(* Logix 5000 project; controller CTRL_PLC_V30 vendor 1 type 14 code 212 rev 34.11; software revision 34.02 *)

TASK MainTask (continuous, watchdog 500 ms) : MainProgram, DataVersturen
TASK SafetyTask (periodic, rate 20 ms, priority 10, watchdog 20 ms, safety) : SafetyProgram

MODULES
   Local : vendor 1 type 14 code 212 (ICP 0, rev 34.11)
      PLC_ETH_CTRL : vendor 1 type 12 code 219 (Ethernet 192.168.1.120, ICP 2, rev 11.1)
      BUSPWR_CTRL : 2198-P208 (Ethernet 192.168.1.18, rev 14.1, A_MotionDiagnostics RPI 1 ms, B_MotionSync RPI 2 ms)
      DRIVER : vendor 1 type 45 code 12 (Ethernet 192.168.1.19, rev 9.3, C_Safety_Output RPI 20 ms, A_MotionDiagnostics RPI 1 ms, B_MotionSync RPI 2 ms, D_Safety_Input RPI 10 ms)
      RIO_CTRL : 1734-AENTR (Ethernet 192.168.1.113, rev 5.17, Output RPI 20 ms)
         Master_IOLINK : vendor 1 type 155 code 1 (PointIO 7, rev 2.1, StandardDataDriven RPI 20 ms)   // 4 channel master IO-link
         INP1_CTRL : 1734-IB4 (PointIO 3, rev 3.1)
         INP2_CTRL : 1734-IB4 (PointIO 4, rev 3.1)
         OUTP2_CTRL : vendor 1 type 7 code 231 (PointIO 6, rev 3.1)
         OUTP1_CTRL : vendor 1 type 7 code 231 (PointIO 5, rev 3.1)
         Safety_OUT : vendor 1 type 35 code 16 (PointIO 2, rev 2.1, Output RPI 20 ms, Input RPI 10 ms)
         Safety_IN : vendor 1 type 35 code 15 (PointIO 1, rev 2.1, Output RPI 20 ms, Input RPI 10 ms)
      @fcc730f7@:Partner : vendor 1 type 14 code 171 (ICP 1, rev 34.11)
END_MODULES

TYPE UDT_COMM_CTRL_TO_SPLC :
STRUCT
   CONTROLLER_STATUS : CONNECTION_STATUS;
   AUX_MCHS_WATCHDOG_CC_BT : BOOL;
   CMD_CCMN_SCLW_RAD_RELEASE_BRAKE : BOOL;
   CMD_CCMN_SWRW_RAD_RELEASE_BRAKE : BOOL;
   CMD_TEST_ABSR_MODULE : BOOL;
   CMD_TEST_ACSR_MODULE : BOOL;
   CMD_TEST_CHAF_MODULE : BOOL;
   CMD_TEST_MODULAR : BOOL;
   CMD_TEST_RBOT_MODULE : BOOL;
   CMD_TEST_RSSR_MODULE : BOOL;
   CMD_TEST_SARB_MODULE : BOOL;
   CMD_TEST_SWSR_MODULE : BOOL;
   CMD_TEST_TBM_MODULE : BOOL;
   QSP_BTDS_XBTDS_DISABLE_LIMITS : BOOL;
   QSP_CCMB_LASERLIGHT_ON : BOOL;
   QSP_CCMF_LASERLIGHT_ON : BOOL;
   QSP_GTCV_ACKNOWLEDGE_MUTE_SCREEN : BOOL;
   QSP_GTRU_TRAV_TO_PICKUP : BOOL;
   QSP_GTRU_TRAV_TO_RELEASE : BOOL;
   QSP_XBDSL_FEEDBACK_FAULT_BRAKE : BOOL;
   QSP_XBDSR_FEEDBACK_FAULT_BRAKE : BOOL;
   QSP_XBTDS_FEEDBACK_FAULT_BRAKE : BOOL;
   QSP_XCCDS_FEEDBACK_FAULT_BRAKE : BOOL;
   QSP_XPBST_FEEDBACK_FAULT_BRAKE : BOOL;
   ZZZ_CC_TO_BT_BOOL_1 : BOOL;
   ZZZ_CC_TO_BT_BOOL_2 : BOOL;
   ZZZ_CC_TO_BT_BOOL_3 : BOOL;
   ZZZ_CC_TO_BT_BOOL_4 : BOOL;
   ZZZ_CC_TO_BT_BOOL_5 : BOOL;
   ZZZ_CC_TO_BT_BOOL_6 : BOOL;
   ZZZ_CC_TO_BT_BOOL_7 : BOOL;
   ZZZ_CC_TO_BT_BOOL_8 : BOOL;
   ZZZ_CC_TO_BT_BOOL_9 : BOOL;
   ZZZ_CC_TO_BT_REAL_1 : REAL;
   ZZZ_CC_TO_BT_REAL_2 : REAL;
   ZZZ_CC_TO_BT_REAL_3 : REAL;
   ZZZ_CC_TO_BT_REAL_4 : REAL;
   ZZZ_CC_TO_BT_REAL_5 : REAL;
END_STRUCT
END_TYPE

TYPE UDT_COMM_SPLC_TO_CTRL :
STRUCT
   CONTROLLER_STATUS : CONNECTION_STATUS;
   AUX_MCHS_WATCHDOG_BT_CC : BOOL;
   CMD_SPLC_IFS_CCAM_STEP_TBM : BOOL;
   FATAL_FAULTS_HWDI : DINT;
   FATAL_FAULTS_HWDI_SIO : DINT;
   FATAL_FAULTS_MCHG : DINT;
   FATAL_FAULTS_MCHS : DINT;
   FATAL_FAULTS_SPLC_ABSR : DINT;
   FATAL_FAULTS_SPLC_ACSR : DINT;
   FATAL_FAULTS_SPLC_BDST : DINT;
   FATAL_FAULTS_SPLC_RSSR : DINT;
   FATAL_FAULTS_SPLC_SARB : DINT;
   FATAL_FAULTS_SPLC_SCCV : DINT;
   FATAL_FAULTS_SPLC_SWSR : DINT;
   FATAL_FAULTS_SPLC_TBM : DINT;
   FCO_HWDI_SYSTEMS_OK_SPLC : BOOL;
   ICF_SPLC_BEAM22_PRESENT : BOOL;
   ICF_SPLC_ROBOT_PREPARED : BOOL;
   ICR_BTDS_NOT_AT_LEFT_POS_LIMIT : BOOL;
   ICR_BTDS_NOT_AT_RIGHT_NEG_LIMIT : BOOL;
   ICR_BTMO_MOTORS_OFF_FEEDBACK : BOOL;
   ICR_CCDS_NOT_AT_LEFT_NEG_LIMIT : BOOL;
   ICR_CCDS_NOT_AT_RIGHT_POS_LIMIT : BOOL;
   IFS_BSMN_1BL2_REWIND_MATERIAL : BOOL;
   IFS_BSMN_1BLO_REWIND_MATERIAL : BOOL;
   IFS_BSMN_2BL2_REWIND_MATERIAL : BOOL;
   IFS_BSMN_2BLO_REWIND_MATERIAL : BOOL;
   IFS_BTAM_STEP : BOOL;
   IFS_CCAM_STEP : BOOL;
   IFS_CSMN_1PLO_REWIND_MATERIAL : BOOL;
   IFS_CSMN_2PLO_REWIND_MATERIAL : BOOL;
   IFS_CSMN_3PLO_REWIND_MATERIAL : BOOL;
   IFS_CSMN_INLO_REWIND_MATERIAL : BOOL;
   IKS_MCHG_CONTROLS_ON : BOOL;
   IPB_BSMN_1BL2_CNV_FEED2 : BOOL;
   IPB_BSMN_2BL2_CNV_FEED : BOOL;
   IPB_CSMN_INCV_FEED_INSIDE : BOOL;
   IPB_CSMN_SWLO_LFT_CNV_FEED2 : BOOL;
   ISP_1BAR_CONNECT_MOTORS : BOOL;
   ISP_1BAR_DRIVE_ENABLE : BOOL;
   ISP_1BCU_SAFETY_DOORS_CLOSED : BOOL;
   ISP_1BCV_CONNECT_MOTORS : BOOL;
   ISP_1BCV_DRIVE_ENABLE : BOOL;
   ISP_1BL2_SAFETY_NOT_ACTIVATED : BOOL;
   ISP_1BLO_SAFETY_NOT_ACTIVATED : BOOL;
   ISP_1PCV_CONNECT_MOTORS : BOOL;
   ISP_1PCV_DRIVE_ENABLE : BOOL;
   ISP_1PLO_SAFETY_NOT_ACTIVATED : BOOL;
   ISP_2BAR_CONNECT_MOTORS : BOOL;
   ISP_2BAR_DRIVE_ENABLE : BOOL;
   ISP_2BCU_SAFETY_DOORS_CLOSED : BOOL;
   ISP_2BCV_CONNECT_MOTORS : BOOL;
   ISP_2BCV_DRIVE_ENABLE : BOOL;
   ISP_2BL2_SAFETY_NOT_ACTIVATED : BOOL;
   ISP_2BLO_SAFETY_NOT_ACTIVATED : BOOL;
   ISP_2PCV_CONNECT_MOTORS : BOOL;
   ISP_2PCV_DRIVE_ENABLE : BOOL;
   ISP_3PCV_CONNECT_MOTORS : BOOL;
   ISP_3PCV_DRIVE_ENABLE : BOOL;
   ISP_2PLO_SAFETY_NOT_ACTIVATED : BOOL;
   ISP_3PLO_SAFETY_NOT_ACTIVATED : BOOL;
   ISP_BDLD_CONNECT_MOTORS : BOOL;
   ISP_BDLD_DRIVE_ENABLE : BOOL;
   ISP_BDLD_LIGHT_CURTAIN_BLOCKED : BOOL;
   ISP_BDLD_RAD_AT_FRONT : BOOL;
   ISP_BDLD_RAD_AT_FRONT_SAFE_AREA : BOOL;
   ISP_BDLD_RAD_AT_MIDDLE : BOOL;
   ISP_BDLD_SAFETY_NOT_ACTIVATED : BOOL;
   ISP_BDSE_INITIALIZE_ARMS : BOOL;
   ISP_BDSE_LFT_CONNECT_MOTORS : BOOL;
   ISP_BDSE_LFT_DRIVE_ENABLE : BOOL;
   ISP_BDSE_RHT_AT_LOAD_AREA : BOOL;
   ISP_BDSE_RHT_CONNECT_MOTORS : BOOL;
   ISP_BDSE_RHT_DRIVE_ENABLE : BOOL;
   ISP_BDST_LOAD_SAFETY_SCR_NOT_TRIPPED : BOOL;
   ISP_BDST_MID_SAFETY_SCR_NOT_TRIPPED : BOOL;
   ISP_BDST_REAR_SAFETY_SCR_NOT_TRIPPED : BOOL;
   ISP_BDST_REAR_SAFETY_SCR_OK : BOOL;
   ISP_BPCA_CONNECT_MOTORS : BOOL;
   ISP_BPCA_DRIVE_ENABLE : BOOL;
   ISP_BPCU_SAFETY_DOOR_CLOSED : BOOL;
   ISP_BPCU_SAFETY_FENCES_CLOSED : BOOL;
   ISP_BPCV_CONNECT_MOTORS : BOOL;
   ISP_BPCV_DRIVE_ENABLE : BOOL;
   ISP_BPSO_CONNECT_MOTORS : BOOL;
   ISP_BPSO_DRIVE_ENABLE : BOOL;
   ISP_BSCV_CONNECT_MOTORS : BOOL;
   ISP_BSCV_DRIVE_ENABLE : BOOL;
   ISP_BTDD_CONNECT_MOTORS : BOOL;
   ISP_BTDD_DRIVE_ENABLE : BOOL;
   ISP_BTDD_RELEASE_BRAKE : BOOL;
   ISP_BTDH_CONNECT_MOTORS : BOOL;
   ISP_BTDH_DRIVE_ENABLE : BOOL;
   ISP_BTDH_RELEASE_BRAKE : BOOL;
   ISP_BTDR_CONNECT_MOTORS : BOOL;
   ISP_BTDR_DRIVE_ENABLE : BOOL;
   ISP_BTDR_RELEASE_BRAKE : BOOL;
   ISP_BTDS_AT_BTTR_AREA : BOOL;
   ISP_BTDS_CONNECT_MOTORS : BOOL;
   ISP_BTDS_DRIVE_ENABLE : BOOL;
   ISP_BTDS_LEFT_LIMIT_OK : BOOL;
   ISP_BTDS_RIGHT_LIMIT_OK : BOOL;
   ISP_BTMN_AREA_ENTRY_NOT_ACTIVE : BOOL;
   ISP_BTMN_BT_DRUM_REL_BRAKE_MODE_ACTIVE : BOOL;
   ISP_BTMN_DOOR_TBM_BR1_SAFETY_NOT_TRIPPED : BOOL;
   ISP_BTMN_DOOR_TBM_BR2_SAFETY_NOT_TRIPPED : BOOL;
   ISP_BTMN_LFT_TRACK_FIRST_RESET_DONE : BOOL;
   ISP_BTMN_LFT_TRACK_SAFETY_NOT_ACTIVATED : BOOL;
   ISP_BTMN_REAR_TRACK_FIRST_RESET_DONE : BOOL;
   ISP_BTMN_REAR_TRACK_SAF_NOT_ACTIVATED : BOOL;
   ISP_BTMN_RHT_TRACK_SAFETY_NOT_ACTIVATED : BOOL;
   ISP_BTMN_TBM_AREA_NOT_ACTIVATED : BOOL;
   ISP_BTMN_TBM_BT_JOG_MODE : BOOL;
   ISP_BTMN_TBM_BT_SHUTTLE_REL_BRAKE_MODE : BOOL;
   ISP_BTMO_RAD_DRIVE_ENABLE : BOOL;
   ISP_BTMO_SAFETY_OVERRULED : BOOL;
   ISP_CCDR_CDAR_CONNECT_MOTORS : BOOL;
   ISP_CCDR_CDRO_CONNECT_MOTORS : BOOL;
   ISP_CCDR_CDTR_CONNECT_MOTORS : BOOL;
   ISP_CCDS_AT_ACSR_POSITION : BOOL;
   ISP_CCDS_CONNECT_MOTORS : BOOL;
   ISP_CCDS_DRIVE_ENABLE : BOOL;
   ISP_CCDS_LEFT_LIMIT_OK : BOOL;
   ISP_CCDS_RIGHT_LIMIT_OK : BOOL;
   ISP_CCMB_SAFETY_OVERRULED : BOOL;
   ISP_CCMC_DRIVE_ENABLE : BOOL;
   ISP_CCMF_CONNECT_MOTORS : BOOL;
   ISP_CCMF_SAFETY_OVERRULED : BOOL;
   ISP_CCMN_BDLD_AREA_NOT_ACTIVATED : BOOL;
   ISP_CCMN_DOOR_TBM_REAR_SAF_NOT_TRIPPED : BOOL;
   ISP_CCMN_FRNT_TRACK_SAFETY_NOT_ACTIVATED : BOOL;
   ISP_CCMN_OPERATOR_AREA_ENTRY_NOT_ACTIVE : BOOL;
   ISP_CCMN_OPERATOR_AREA_NOT_ACTIVATED : BOOL;
   ISP_CCMN_REAR_TRACK_FIRST_RESET_DONE : BOOL;
   ISP_CCMN_REAR_TRACK_SAF_NOT_ACTIVATED : BOOL;
   ISP_CCMN_TBM_AREA_ENTRY_NOT_ACTIVE : BOOL;
   ISP_CCMN_TBM_AREA_NOT_ACTIVATED : BOOL;
   ISP_CCMN_TBM_CC_JOG_MODE : BOOL;
   ISP_CCMN_TBM_CC_SHUTTLE_REL_BRAKE_MODE : BOOL;
   ISP_CCMR_DRIVE_ENABLE : BOOL;
   ISP_CCMT_DRIVE_ENABLE : BOOL;
   ISP_CDAR_DRIVE_ENABLE : BOOL;
   ISP_CDRO_DRIVE_ENABLE : BOOL;
   ISP_CDTR_DRIVE_ENABLE : BOOL;
   ISP_CENT_BT_SAFETY_OK : BOOL;
   ISP_CENT_CC_SAFETY_OK : BOOL;
   ISP_CWLO_FEST_SAFETY_DOOR_CLOSED : BOOL;
   ISP_CWLO_LFT_STRIP_NOT_SELECTED : BOOL;
   ISP_CWLO_RHT_STRIP_NOT_SELECTED : BOOL;
   ISP_CWLO_SAFETY_DOOR_CLOSED : BOOL;
   ISP_CWTC_CONNECT_MOTORS : BOOL;
   S_ISP_CWTC_DRIVE_ENABLE : BOOL;
   ISP_E_STOP_ACTIVATED : BOOL;
   ISP_GTCV_EJECTION_TABLE_UP : BOOL;
   ISP_GTRU_CONNECT_MOTORS : BOOL;
   ISP_GTRU_DRIVE_ENABLE : BOOL;
   ISP_GTRU_GRIPPER_OPEN : BOOL;
   ISP_GTRU_LIGHT_CURTAIN_BLOCKED : BOOL;
   ISP_GTRU_RAD_AT_FRONT : BOOL;
   ISP_GTRU_SAFETY_MUTE_ACTIVE : BOOL;
   ISP_GTRU_SAFETY_NOT_ACTIVATED : BOOL;
   ISP_GTRU_TIRE_DETECTED : BOOL;
   ISP_GTRU_TRAV_AT_PICKUP : BOOL;
   ISP_GTRU_TRAV_AT_RELEASE : BOOL;
   ISP_INCV_CONNECT_MOTORS : BOOL;
   ISP_INCV_DRIVE_ENABLE : BOOL;
   ISP_INLO_SAFETY_NOT_ACTIVATED : BOOL;
   ISP_MAIN_PRESSURE_PRESENT : BOOL;
   ISP_PACU_SAFETY_DOOR_CLOSED : BOOL;
   ISP_PACU_SAFETY_FENCES_CLOSED : BOOL;
   ISP_PACV_CONNECT_MOTORS : BOOL;
   ISP_PACV_DRIVE_ENABLE : BOOL;
   ISP_PBCV_CONNECT_MOTORS : BOOL;
   ISP_PBCV_DRIVE_ENABLE : BOOL;
   ISP_PBCV_SAFETY_DOORS_CLOSED : BOOL;
   ISP_PBST_CONNECT_MOTORS : BOOL;
   ISP_PBST_DRIVE_ENABLE : BOOL;
   ISP_PBUD_CONNECT_MOTORS : BOOL;
   ISP_PBUD_DRIVE_ENABLE : BOOL;
   ISP_PBUD_SAFE_SPD_TRIPPED : BOOL;
   ISP_RBCL_CONNECT_MOTORS : BOOL;
   ISP_RBCL_DRIVE_ENABLE : BOOL;
   ISP_RBOT_ENABLE : BOOL;
   ISP_RSLC_CONNECT_MOTORS : BOOL;
   ISP_RSLC_DRIVE_ENABLE : BOOL;
   ISP_RSLO_REAR_SAFETY_NOT_ACTIVATED : BOOL;
   ISP_RSLO_SIDE_SAFETY_NOT_ACTIVATED : BOOL;
   ISP_RSLW_AT_LETOFF_AREA : BOOL;
   ISP_RSLW_CONNECT_MOTORS : BOOL;
   ISP_RSLW_DRIVE_ENABLE : BOOL;
   ISP_RSLW_RAD_CONNECT_MOTORS : BOOL;
   ISP_RSLW_RAD_DRIVE_ENABLE : BOOL;
   ISP_RSLW_TRAV_CONNECT_MOTORS : BOOL;
   ISP_RSLW_TRAV_DRIVE_ENABLE : BOOL;
   ISP_RSMN_JOG_MODE : BOOL;
   ISP_RSMN_RS_INSIDE_FIRST_RESET_DONE : BOOL;
   ISP_RSMN_RSLO_JOG_MODE : BOOL;
   ISP_RSMN_RSLO_LFT_JOG_MODE : BOOL;
   ISP_RSMN_RSLO_RHT_JOG_MODE : BOOL;
   ISP_RSMN_RSXR_REL_BRAKE_MODE : BOOL;
   ISP_RSMN_TBM_AREA_SAFETY_NOT_ACTIVE : BOOL;
   ISP_RSRC_CONNECT_MOTORS : BOOL;
   ISP_RSRC_DRIVE_ENABLE : BOOL;
   ISP_RSRW_CONNECT_MOTORS : BOOL;
   ISP_RSRW_DRIVE_ENABLE : BOOL;
   ISP_RSRW_RAD_CONNECT_MOTORS : BOOL;
   ISP_RSRW_RAD_DRIVE_ENABLE : BOOL;
   ISP_RSRW_TRAV_CONNECT_MOTORS : BOOL;
   ISP_RSRW_TRAV_DRIVE_ENABLE : BOOL;
   ISP_SARB_ENABLE : BOOL;
   ISP_SCLW_AT_LETOFF_AREA : BOOL;
   ISP_SCLW_CONNECT_MOTORS : BOOL;
   ISP_SCLW_DRIVE_ENABLE : BOOL;
   ISP_SCLW_RAD_CONNECT_MOTORS : BOOL;
   ISP_SCLW_RAD_DRIVE_ENABLE : BOOL;
   ISP_SCLW_TRAV_CONNECT_MOTORS : BOOL;
   ISP_SCLW_TRAV_DRIVE_ENABLE : BOOL;
   ISP_SCMN_JOG_MODE : BOOL;
   ISP_SCMN_RELEASE_SCXR_BRAKE : BOOL;
   ISP_SCMN_SC_INSIDE_FIRST_RESET_DONE : BOOL;
   ISP_SCMN_TBM_AREA_SAFETY_NOT_ACTIVE : BOOL;
   ISP_SCRW_CONNECT_MOTORS : BOOL;
   ISP_SCRW_DRIVE_ENABLE : BOOL;
   ISP_SCRW_RAD_CONNECT_MOTORS : BOOL;
   ISP_SCRW_RAD_DRIVE_ENABLE : BOOL;
   ISP_SCRW_TRAV_CONNECT_MOTORS : BOOL;
   ISP_SCRW_TRAV_DRIVE_ENABLE : BOOL;
   ISP_SLOW_START_PRESSURE_NOT_OK : BOOL;
   ISP_SPLC_FAULT_EXISTS : BOOL;
   ISP_SPLC_REAR_TRACK_SAFETY_RST_INITIATED : BOOL;
   ISP_SPLC_SAFETY_SIGNATURE_EXISTS : BOOL;
   ISP_SPLC_TBM_BT_AREA_ENTRY_OK_DELAY : BOOL;
   ISP_SPLC_TBM_BT_LC_OK_DELAY : BOOL;
   ISP_SPLC_TBM_CC_AREA_ENTRY_OPER_OK_DELAY : BOOL;
   ISP_SPLC_TBM_CC_AREA_ENTRY_TBM_OK_DELAY : BOOL;
   ISP_SPLC_TBM_CC_LC_OPER_OK_DELAY : BOOL;
   ISP_SPLC_TBM_CC_LC_TBM_OK_DELAY : BOOL;
   ISP_SWL2_SAFETY_NOT_ACTIVATED : BOOL;
   ISP_SWL3_REAR_SAFETY_NOT_ACTIVATED : BOOL;
   ISP_SWL3_SIDE_SAFETY_NOT_ACTIVATED : BOOL;
   ISP_SWLC_CONNECT_MOTORS : BOOL;
   ISP_SWLC_DRIVE_ENABLE : BOOL;
   ISP_SWLO_INSIDE_SAFETY_NOT_ACTIVE : BOOL;
   ISP_SWLO_SAFETY_NOT_ACTIVATED : BOOL;
   ISP_SWLW_AT_LETOFF_AREA : BOOL;
   ISP_SWLW_CONNECT_MOTORS : BOOL;
   ISP_SWLW_DRIVE_ENABLE : BOOL;
   ISP_SWLW_RAD_CONNECT_MOTORS : BOOL;
   ISP_SWLW_RAD_DRIVE_ENABLE : BOOL;
   ISP_SWLW_TRAV_CONNECT_MOTORS : BOOL;
   ISP_SWLW_TRAV_DRIVE_ENABLE : BOOL;
   ISP_SWMN_JOG_MODE : BOOL;
   ISP_SWMN_SW_INSIDE_FIRST_RESET_DONE : BOOL;
   ISP_SWMN_SWL3_JOG_MODE : BOOL;
   ISP_SWMN_SWL3_LFT_JOG_MODE : BOOL;
   ISP_SWMN_SWL3_RHT_JOG_MODE : BOOL;
   ISP_SWMN_SWLC_DOOR_CLOSED : BOOL;
   ISP_SWMN_RELEASE_SWXR_BRAKE : BOOL;
   ISP_SWMN_TBM_AREA_SAFETY_NOT_ACTIVE : BOOL;
   ISP_SWRC_CONNECT_MOTORS : BOOL;
   ISP_SWRC_DRIVE_ENABLE : BOOL;
   ISP_SWRW_CONNECT_MOTORS : BOOL;
   ISP_SWRW_DRIVE_ENABLE : BOOL;
   ISP_SWRW_RAD_CONNECT_MOTORS : BOOL;
   ISP_SWRW_RAD_DRIVE_ENABLE : BOOL;
   ISP_SWRW_TRAV_CONNECT_MOTORS : BOOL;
   ISP_SWRW_TRAV_DRIVE_ENABLE : BOOL;
   ISP_TDAR_CONNECT_MOTORS : BOOL;
   ISP_TDAR_DRIVE_ENABLE : BOOL;
   ISP_TDCU_SAFETY_COVER_CLOSED : BOOL;
   ISP_TDCV_CONNECT_MOTORS : BOOL;
   ISP_TDCV_DRIVE_ENABLE : BOOL;
   ISP_TDLO_LFT_SAFETY_NOT_ACTIVATED : BOOL;
   ISP_TDLO_RHT_SAFETY_NOT_ACTIVATED : BOOL;
   ISP_TDLO_SAFETY_NOT_ACTIVATED : BOOL;
   ISP_TEST_MODE_SELECTED : BOOL;
   ISP_TPGU_SAFETY_OVERRULED : BOOL;
   ISS_BSMN_1BL2_WINDOFF : BOOL;
   ISS_BSMN_1BL2_WINDUP : BOOL;
   ISS_BSMN_1BLO_WINDOFF : BOOL;
   ISS_BSMN_1BLO_WINDUP : BOOL;
   ISS_BSMN_2BL2_WINDOFF : BOOL;
   ISS_BSMN_2BL2_WINDUP : BOOL;
   ISS_BSMN_2BLO_WINDOFF : BOOL;
   ISS_BSMN_2BLO_WINDUP : BOOL;
   ISS_CSMN_1PLO_WINDOFF : BOOL;
   ISS_CSMN_1PLO_WINDUP : BOOL;
   ISS_CSMN_2PLO_WINDOFF : BOOL;
   ISS_CSMN_2PLO_WINDUP : BOOL;
   ISS_CSMN_3PLO_WINDOFF : BOOL;
   ISS_CSMN_3PLO_WINDUP : BOOL;
   ISS_CSMN_INLO_WINDOFF : BOOL;
   ISS_CSMN_INLO_WINDUP : BOOL;
   ISS_CSMN_SWL2_LFT_WINDOFF : BOOL;
   ISS_CSMN_SWL2_LFT_WINDUP : BOOL;
   ISS_CSMN_SWL2_RHT_WINDOFF : BOOL;
   ISS_CSMN_SWL2_RHT_WINDUP : BOOL;
   ISS_CSMN_SWL2_WINDOFF : BOOL;
   ISS_CSMN_SWL2_WINDUP : BOOL;
   ISS_CSMN_SWLO_LFT_WINDOFF : BOOL;
   ISS_CSMN_SWLO_LFT_WINDUP : BOOL;
   ISS_CSMN_SWLO_RHT_WINDOFF : BOOL;
   ISS_CSMN_SWLO_RHT_WINDUP : BOOL;
   ISS_CSMN_SWLO_WINDOFF : BOOL;
   ISS_CSMN_SWLO_WINDUP : BOOL;
   ISS_RSMN_RSLW_JOG_FWD : BOOL;
   ISS_RSMN_RSLW_JOG_REV : BOOL;
   ISS_RSMN_RSRW_JOG_FWD : BOOL;
   ISS_RSMN_RSRW_JOG_REV : BOOL;
   ISS_SCMN_SCLW_JOG_FWD : BOOL;
   ISS_SCMN_SCLW_JOG_REV : BOOL;
   ISS_SCMN_SCRW_JOG_FWD : BOOL;
   ISS_SCMN_SCRW_JOG_REV : BOOL;
   ISS_SWMN_SWLW_JOG_FWD : BOOL;
   ISS_SWMN_SWLW_JOG_REV : BOOL;
   ISS_SWMN_SWRW_JOG_FWD : BOOL;
   ISS_SWMN_SWRW_JOG_REV : BOOL;
   ISS_TDMN_TDLO_LFT_WINDOFF : BOOL;
   ISS_TDMN_TDLO_LFT_WINDUP : BOOL;
   ISS_TDMN_TDLO_RHT_WINDOFF : BOOL;
   ISS_TDMN_TDLO_RHT_WINDUP : BOOL;
   ISS_TDMN_TDLO_WINDOFF : BOOL;
   ISS_TDMN_TDLO_WINDUP : BOOL;
   ISP_XXMN_DOOR_ACSR_XX_CLOSED : BOOL;
   ISP_XXMN_DOOR_SC_XX_CLOSED : BOOL;
   ISP_XXMN_DOOR_XX_TBM_CLOSED : BOOL;
   ISP_XXMN_INSIDE_SAFETY_BTTR_RESET_REQ : BOOL;
   ZZZ_BT_TO_CC_BOOL_1 : BOOL;
   ZZZ_BT_TO_CC_BOOL_2 : BOOL;
   ZZZ_BT_TO_CC_BOOL_3 : BOOL;
   ZZZ_BT_TO_CC_BOOL_4 : BOOL;
   ZZZ_BT_TO_CC_BOOL_5 : BOOL;
   ZZZ_BT_TO_CC_BOOL_6 : BOOL;
   ZZZ_BT_TO_CC_BOOL_7 : BOOL;
   ZZZ_BT_TO_CC_BOOL_8 : BOOL;
   ZZZ_BT_TO_CC_BOOL_9 : BOOL;
   ZZZ_BT_TO_CC_REAL_1 : REAL;
   ZZZ_BT_TO_CC_REAL_2 : REAL;
   ZZZ_BT_TO_CC_REAL_3 : REAL;
   ZZZ_BT_TO_CC_REAL_4 : REAL;
   ZZZ_BT_TO_CC_REAL_5 : REAL;
   ISS_BSMN_1BLO_DRIVE_ROLLS_TO_REST : BOOL;
   ISS_BSMN_1BLO_DRIVE_ROLLS_ENGAGE : BOOL;
   ISP_1BLO_TWO_HAND_OVERRIDE : BOOL;
   ISS_BSMN_1BLO_CART_LOCK : BOOL;
   ISS_BSMN_1BLO_CART_UNLOCK : BOOL;
   ISS_BSMN_2BLO_DRIVE_ROLLS_TO_REST : BOOL;
   ISS_BSMN_2BLO_DRIVE_ROLLS_ENGAGE : BOOL;
   ISP_2BLO_TWO_HAND_OVERRIDE : BOOL;
   ISS_BSMN_2BLO_CART_LOCK : BOOL;
   ISS_BSMN_2BLO_CART_UNLOCK : BOOL;
   ISS_TDMN_TDLO_DRIVE_ROLLS_ENGAGE : BOOL;
   ISS_TDMN_TDLO_DRIVE_ROLLS_TO_REST : BOOL;
   ISP_TDLO_TWO_HAND_OVERRIDE : BOOL;
   ISS_TDMN_TDLO_CART_LOCK : BOOL;
   ISS_TDMN_TDLO_CART_UNLOCK : BOOL;
   ISS_SWLO_RHT_DRIVE_ROLLS_REST : BOOL;
   ISS_SWLO_RHT_DRIVE_ROLLS_ENGAGE : BOOL;
   ISS_CSMN_SWLO_RHT_CART_LOCK : BOOL;
   ISS_CSMN_SWLO_RHT_CART_UNLOCK : BOOL;
   ISP_SWLO_RHT_TWO_HAND_OVERRIDE : BOOL;
   ISS_SWLO_LFT_DRIVE_ROLLS_REST : BOOL;
   ISS_SWLO_LFT_DRIVE_ROLLS_ENGAGE : BOOL;
   ISS_CSMN_SWLO_LFT_CART_LOCK : BOOL;
   ISS_CSMN_SWLO_LFT_CART_UNLOCK : BOOL;
   ISP_SWLO_LFT_TWO_HAND_OVERRIDE : BOOL;
END_STRUCT
END_TYPE

VAR_GLOBAL   (* controller tags *)
   Aantal_RondjesT1 : DINT := 40;
   Aantal_RondjesT2 : DINT;
   As_Test1_CTRL : AXIS_CIP_DRIVE;
   As_Test2_CTRL : AXIS_CIP_DRIVE;
   AsTest1Accel : REAL := 1000000.0;
   AsTest1Snelheid : REAL := 3500.0;
   AsTest1StartPos : REAL;
   AsTest1StopPos : REAL := 9500.0;
   AsTest2Accel : REAL;
   AsTest2Snelheid : REAL;
   AsTest2StartPos : REAL;
   AsTest2StopPos : REAL;
   BOOL : BOOL;
   Control_Volt_Van_SAF : BOOL;
   Drive1 : MOTION_GROUP;
   Drive_SAFE_OFF1 : ALIAS FOR DRIVER:SO.SafeTorqueOff1;
   Drive_SAFE_OFF2 : ALIAS FOR DRIVER:SO.SafeTorqueOff2;
   ERROR : BOOL;
   ERROR_1 : BOOL := 1;
   ERROR_2 : BOOL := 1;
   ESTP_ACTIVATED : BOOL;
   HomeT1 : ALIAS FOR IOP_HMI_BT[0].2;
   HomeT2 : ALIAS FOR IOP_HMI_BT[1].2;
   ILB_RESET_SAFETY1 : BOOL := 1;
   ILG_CTRL_VOLT1 : BOOL;
   IO_CTRL_TO_SPLC : UDT_COMM_CTRL_TO_SPLC := (CONTROLLER_STATUS.RunMode := 1); {produced}
   IO_SPLC_TO_CTRL : UDT_COMM_SPLC_TO_CTRL;
   IOP_HMI_BT : DINT[2];
   IOP_HMI_REAL : REAL[20] := ([0] := 3500.0, [1] := 1000000.0, [3] := 9500.0, [4] := 40.0);
   MDA_DATACHOICE : INT := 2;
   MDB_DATACHOICE : INT := 2;
   Motionback : MOTION_INSTRUCTION;
   Motionback2 : MOTION_INSTRUCTION;
   Motioncontrol13 : MOTION_INSTRUCTION := (FLAGS := -1845493760, EN := 1, ER := 1, ERR := 13, EXERR := 6);
   Motioncontrol14 : MOTION_INSTRUCTION := (FLAGS := -1845493760, EN := 1, ER := 1, ERR := 13, EXERR := 6);
   Motioncontrol20 : MOTION_INSTRUCTION;
   Motioncontrol21 : MOTION_INSTRUCTION := (FLAGS := -1476395008, EN := 1, DN := 1, PC := 1, STATE := 17);
   Motioncontrol26 : MOTION_INSTRUCTION := (FLAGS := -1442840576, EN := 1, DN := 1, PC := 1, STATE := 17); {access None}
   Motioncontrol27 : MOTION_INSTRUCTION := (FLAGS := -1442840576, EN := 1, DN := 1, PC := 1, STATE := 17);
   Motioncontrol3 : MOTION_INSTRUCTION := (FLAGS := -1442840576, EN := 1, DN := 1, PC := 1);
   Motioncontrol30 : MOTION_INSTRUCTION := (FLAGS := 33554432);
   Motioncontrol31 : MOTION_INSTRUCTION;
   Motioncontrol4 : MOTION_INSTRUCTION := (FLAGS := -1442840576, EN := 1, DN := 1, PC := 1);
   Motionctrl1 : MOTION_INSTRUCTION := (FLAGS := -1577058304, EN := 1, DN := 1, STATE := 1);
   Motionctrl2 : MOTION_INSTRUCTION := (FLAGS := -1577058304, EN := 1, DN := 1, STATE := 1);
   Motionstart1 : MOTION_INSTRUCTION := (FLAGS := -1845493760, EN := 1, ER := 1, ERR := 20);
   Motionstartl2 : MOTION_INSTRUCTION := (FLAGS := -1845493760, EN := 1, ER := 1, ERR := 20);
   Motionstop1 : MOTION_INSTRUCTION;
   Motionstop2 : MOTION_INSTRUCTION;
   OvertravelFault : BOOL; {access None}
   OvertravelFault2 : BOOL; {access None}
   Powersupply_1 : AXIS_CIP_DRIVE;
   QOP_HMI_BT : DINT[10] := ([0] := 6272);
   QOP_HMI_GRAPH1_HDR : REAL[10] := ([3] := 9500.0, [5] := 30.053297, [6] := 20.0, [7] := 1.0); {access Read Only}
        [2]   // Xmin
        [3]   // Xmax
        [7]   // Ywaarders per gridline
        [6]   // Xwaardes per gridline
        [4]   // Ymin
        [5]   // Ymax
   QOP_HMI_GRAPH1_LINE1_DATAX : REAL[800] := ([0] := 0.1, [1] := 11.975, [2] := 23.85, [3] := 35.725, [4] := 47.6, [5] := 59.475, [6] := 71.35, [7] := 83.225, [8] := 95.1, [9] := 106.975, [10] := 118.85, [11] := 130.725, [12] := 142.6, [13] := 154.475, [14] := 166.35, [15] := 178.225, [16] := 190.1, [17] := 201.975, [18] := 213.85, [19] := 225.725, [20] := 237.6, [21] := 249.475, [22] := 261.35, [23] := 273.225, [24] := 285.1, [25] := 296.975, [26] := 308.85, [27] := 320.725, [28] := 332.6, [29] := 344.475, [30] := 356.35, [31] := 368.225, [32] := 380.1, [33] := 391.975, [34] := 403.85, [35] := 415.725, [36] := 427.6, [37] := 439.475, [38] := 451.35, [39] := 463.225, [40] := 475.1, [41] := 486.975, [42] := 498.85, [43] := 510.725, [44] := 522.6, [45] := 534.475, [46] := 546.35, [47] := 558.225, [48] := 570.1, [49] := 581.975, [50] := 593.85, [51] := 605.725, [52] := 617.6, [53] := 629.475, [54] := 641.35, [55] := 653.225, [56] := 665.1, [57] := 676.975, [58] := 688.85, [59] := 700.725,
        [60] := 712.6, [61] := 724.475, [62] := 736.35, [63] := 748.225, [64] := 760.1, [65] := 771.975, [66] := 783.85, [67] := 795.725, [68] := 807.6, [69] := 819.475, [70] := 831.35, [71] := 843.225, [72] := 855.1, [73] := 866.975, [74] := 878.85, [75] := 890.725, [76] := 902.6, [77] := 914.475, [78] := 926.35, [79] := 938.225, [80] := 950.1, [81] := 961.975, [82] := 973.85, [83] := 985.725, [84] := 997.6, [85] := 1009.475, [86] := 1021.35, [87] := 1033.225, [88] := 1045.1, [89] := 1056.975, [90] := 1068.85, [91] := 1080.725, [92] := 1092.6, [93] := 1104.475, [94] := 1116.35, [95] := 1128.225, [96] := 1140.1, [97] := 1151.975, [98] := 1163.85, [99] := 1175.725, [100] := 1187.6, [101] := 1199.475, [102] := 1211.35, [103] := 1223.225, [104] := 1235.1, [105] := 1246.975, [106] := 1258.85, [107] := 1270.725, [108] := 1282.6, [109] := 1294.475, [110] := 1306.35, [111] := 1318.225, [112] := 1330.1, [113] := 1341.975, [114] := 1353.85, [115] := 1365.725, [116] := 1377.6, [117] := 1389.475, [118] := 1401.35, [119] := 1413.225,
        [120] := 1425.1, [121] := 1436.975, [122] := 1448.85, [123] := 1460.725, [124] := 1472.6, [125] := 1484.475, [126] := 1496.35, [127] := 1508.225, [128] := 1520.1, [129] := 1531.975, [130] := 1543.85, [131] := 1555.725, [132] := 1567.6, [133] := 1579.475, [134] := 1591.35, [135] := 1603.225, [136] := 1615.1, [137] := 1626.975, [138] := 1638.85, [139] := 1650.725, [140] := 1662.6, [141] := 1674.475, [142] := 1686.35, [143] := 1698.225, [144] := 1710.1, [145] := 1721.975, [146] := 1733.85, [147] := 1745.725, [148] := 1757.6, [149] := 1769.475, [150] := 1781.35, [151] := 1793.225, [152] := 1805.1, [153] := 1816.975, [154] := 1828.85, [155] := 1840.725, [156] := 1852.6, [157] := 1864.475, [158] := 1876.35, [159] := 1888.225, [160] := 1900.1, [161] := 1911.975, [162] := 1923.85, [163] := 1935.725, [164] := 1947.6, [165] := 1959.475, [166] := 1971.35, [167] := 1983.225, [168] := 1995.1, [169] := 2006.975, [170] := 2018.85, [171] := 2030.725, [172] := 2042.6, [173] := 2054.475, [174] := 2066.35, [175] := 2078.225, [176] := 2090.1, [177] := 2101.975, [178] := 2113.85, [179] := 2125.725,
        [180] := 2137.6, [181] := 2149.475, [182] := 2161.35, [183] := 2173.225, [184] := 2185.1, [185] := 2196.975, [186] := 2208.85, [187] := 2220.725, [188] := 2232.6, [189] := 2244.475, [190] := 2256.35, [191] := 2268.225, [192] := 2280.1, [193] := 2291.975, [194] := 2303.85, [195] := 2315.725, [196] := 2327.6, [197] := 2339.475, [198] := 2351.35, [199] := 2363.225, [200] := 2375.1, [201] := 2386.975, [202] := 2398.85, [203] := 2410.725, [204] := 2422.6, [205] := 2434.475, [206] := 2446.35, [207] := 2458.225, [208] := 2470.1, [209] := 2481.975, [210] := 2493.85, [211] := 2505.725, [212] := 2517.6, [213] := 2529.475, [214] := 2541.35, [215] := 2553.225, [216] := 2565.1, [217] := 2576.975, [218] := 2588.85, [219] := 2600.725, [220] := 2612.6, [221] := 2624.475, [222] := 2636.35, [223] := 2648.225, [224] := 2660.1, [225] := 2671.975, [226] := 2683.85, [227] := 2695.725, [228] := 2707.6, [229] := 2719.475, [230] := 2731.35, [231] := 2743.225, [232] := 2755.1, [233] := 2766.975, [234] := 2778.85, [235] := 2790.725, [236] := 2802.6, [237] := 2814.475, [238] := 2826.35, [239] := 2838.225,
        [240] := 2850.1, [241] := 2861.975, [242] := 2873.85, [243] := 2885.725, [244] := 2897.6, [245] := 2909.475, [246] := 2921.35, [247] := 2933.225, [248] := 2945.1, [249] := 2956.975, [250] := 2968.85, [251] := 2980.725, [252] := 2992.6, [253] := 3004.475, [254] := 3016.35, [255] := 3028.225, [256] := 3040.1, [257] := 3051.975, [258] := 3063.85, [259] := 3075.725, [260] := 3087.6, [261] := 3099.475, [262] := 3111.35, [263] := 3123.225, [264] := 3135.1, [265] := 3146.975, [266] := 3158.85, [267] := 3170.725, [268] := 3182.6, [269] := 3194.475, [270] := 3206.35, [271] := 3218.225, [272] := 3230.1, [273] := 3241.975, [274] := 3253.85, [275] := 3265.725, [276] := 3277.6, [277] := 3289.475, [278] := 3301.35, [279] := 3313.225, [280] := 3325.1, [281] := 3336.975, [282] := 3348.85, [283] := 3360.725, [284] := 3372.6, [285] := 3384.475, [286] := 3396.35, [287] := 3408.225, [288] := 3420.1, [289] := 3431.975, [290] := 3443.85, [291] := 3455.725, [292] := 3467.6, [293] := 3479.475, [294] := 3491.35, [295] := 3503.225, [296] := 3515.1, [297] := 3526.975, [298] := 3538.85, [299] := 3550.725,
        [300] := 3562.6, [301] := 3574.475, [302] := 3586.35, [303] := 3598.225, [304] := 3610.1, [305] := 3621.975, [306] := 3633.85, [307] := 3645.725, [308] := 3657.6, [309] := 3669.475, [310] := 3681.35, [311] := 3693.225, [312] := 3705.1, [313] := 3716.975, [314] := 3728.85, [315] := 3740.725, [316] := 3752.6, [317] := 3764.475, [318] := 3776.35, [319] := 3788.225, [320] := 3800.1, [321] := 3811.975, [322] := 3823.85, [323] := 3835.725, [324] := 3847.6, [325] := 3859.475, [326] := 3871.35, [327] := 3883.225, [328] := 3895.1, [329] := 3906.975, [330] := 3918.85, [331] := 3930.725, [332] := 3942.6, [333] := 3954.475, [334] := 3966.35, [335] := 3978.225, [336] := 3990.1, [337] := 4001.975, [338] := 4013.85, [339] := 4025.725, [340] := 4037.6, [341] := 4049.475, [342] := 4061.35, [343] := 4073.225, [344] := 4085.1, [345] := 4096.975, [346] := 4108.85, [347] := 4120.725, [348] := 4132.6, [349] := 4144.475, [350] := 4156.35, [351] := 4168.225, [352] := 4180.1, [353] := 4191.975, [354] := 4203.85, [355] := 4215.725, [356] := 4227.6, [357] := 4239.475, [358] := 4251.35, [359] := 4263.225,
        [360] := 4275.1, [361] := 4286.975, [362] := 4298.85, [363] := 4310.725, [364] := 4322.6, [365] := 4334.475, [366] := 4346.35, [367] := 4358.225, [368] := 4370.1, [369] := 4381.975, [370] := 4393.85, [371] := 4405.725, [372] := 4417.6, [373] := 4429.475, [374] := 4441.35, [375] := 4453.225, [376] := 4465.1, [377] := 4476.975, [378] := 4488.85, [379] := 4500.725, [380] := 4512.6, [381] := 4524.475, [382] := 4536.35, [383] := 4548.225, [384] := 4560.1, [385] := 4571.975, [386] := 4583.85, [387] := 4595.725, [388] := 4607.6, [389] := 4619.475, [390] := 4631.35, [391] := 4643.225, [392] := 4655.1, [393] := 4666.975, [394] := 4678.85, [395] := 4690.725, [396] := 4702.6, [397] := 4714.475, [398] := 4726.35, [399] := 4738.225, [400] := 4750.1, [401] := 4761.975, [402] := 4773.85, [403] := 4785.725, [404] := 4797.6, [405] := 4809.475, [406] := 4821.35, [407] := 4833.225, [408] := 4845.1, [409] := 4856.975, [410] := 4868.85, [411] := 4880.725, [412] := 4892.6, [413] := 4904.475, [414] := 4916.35, [415] := 4928.225, [416] := 4940.1, [417] := 4951.975, [418] := 4963.85, [419] := 4975.725,
        [420] := 4987.6, [421] := 4999.475, [422] := 5011.35, [423] := 5023.225, [424] := 5035.1, [425] := 5046.975, [426] := 5058.85, [427] := 5070.725, [428] := 5082.6, [429] := 5094.475, [430] := 5106.35, [431] := 5118.225, [432] := 5130.1, [433] := 5141.975, [434] := 5153.85, [435] := 5165.725, [436] := 5177.6, [437] := 5189.475, [438] := 5201.35, [439] := 5213.225, [440] := 5225.1, [441] := 5236.975, [442] := 5248.85, [443] := 5260.725, [444] := 5272.6, [445] := 5284.475, [446] := 5296.35, [447] := 5308.225, [448] := 5320.1, [449] := 5331.975, [450] := 5343.85, [451] := 5355.725, [452] := 5367.6, [453] := 5379.475, [454] := 5391.35, [455] := 5403.225, [456] := 5415.1, [457] := 5426.975, [458] := 5438.85, [459] := 5450.725, [460] := 5462.6, [461] := 5474.475, [462] := 5486.35, [463] := 5498.225, [464] := 5510.1, [465] := 5521.975, [466] := 5533.85, [467] := 5545.725, [468] := 5557.6, [469] := 5569.475, [470] := 5581.35, [471] := 5593.225, [472] := 5605.1, [473] := 5616.975, [474] := 5628.85, [475] := 5640.725, [476] := 5652.6, [477] := 5664.475, [478] := 5676.35, [479] := 5688.225,
        [480] := 5700.1, [481] := 5711.975, [482] := 5723.85, [483] := 5735.725, [484] := 5747.6, [485] := 5759.475, [486] := 5771.35, [487] := 5783.225, [488] := 5795.1, [489] := 5806.975, [490] := 5818.85, [491] := 5830.725, [492] := 5842.6, [493] := 5854.475, [494] := 5866.35, [495] := 5878.225, [496] := 5890.1, [497] := 5901.975, [498] := 5913.85, [499] := 5925.725, [500] := 5937.6, [501] := 5949.475, [502] := 5961.35, [503] := 5973.225, [504] := 5985.1, [505] := 5996.975, [506] := 6008.85, [507] := 6020.725, [508] := 6032.6, [509] := 6044.475, [510] := 6056.35, [511] := 6068.225, [512] := 6080.1, [513] := 6091.975, [514] := 6103.85, [515] := 6115.725, [516] := 6127.6, [517] := 6139.475, [518] := 6151.35, [519] := 6163.225, [520] := 6175.1, [521] := 6186.975, [522] := 6198.85, [523] := 6210.725, [524] := 6222.6, [525] := 6234.475, [526] := 6246.35, [527] := 6258.225, [528] := 6270.1, [529] := 6281.975, [530] := 6293.85, [531] := 6305.725, [532] := 6317.6, [533] := 6329.475, [534] := 6341.35, [535] := 6353.225, [536] := 6365.1, [537] := 6376.975, [538] := 6388.85, [539] := 6400.725,
        [540] := 6412.6, [541] := 6424.475, [542] := 6436.35, [543] := 6448.225, [544] := 6460.1, [545] := 6471.975, [546] := 6483.85, [547] := 6495.725, [548] := 6507.6, [549] := 6519.475, [550] := 6531.35, [551] := 6543.225, [552] := 6555.1, [553] := 6566.975, [554] := 6578.85, [555] := 6590.725, [556] := 6602.6, [557] := 6614.475, [558] := 6626.35, [559] := 6638.225, [560] := 6650.1, [561] := 6661.975, [562] := 6673.85, [563] := 6685.725, [564] := 6697.6, [565] := 6709.475, [566] := 6721.35, [567] := 6733.225, [568] := 6745.1, [569] := 6756.975, [570] := 6768.85, [571] := 6780.725, [572] := 6792.6, [573] := 6804.475, [574] := 6816.35, [575] := 6828.225, [576] := 6840.1, [577] := 6851.975, [578] := 6863.85, [579] := 6875.725, [580] := 6887.6, [581] := 6899.475, [582] := 6911.35, [583] := 6923.225, [584] := 6935.1, [585] := 6946.975, [586] := 6958.85, [587] := 6970.725, [588] := 6982.6, [589] := 6994.475, [590] := 7006.35, [591] := 7018.225, [592] := 7030.1, [593] := 7041.975, [594] := 7053.85, [595] := 7065.725, [596] := 7077.6, [597] := 7089.475, [598] := 7101.35, [599] := 7113.225,
        [600] := 7125.1, [601] := 7136.975, [602] := 7148.85, [603] := 7160.725, [604] := 7172.6, [605] := 7184.475, [606] := 7196.35, [607] := 7208.225, [608] := 7220.1, [609] := 7231.975, [610] := 7243.85, [611] := 7255.725, [612] := 7267.6, [613] := 7279.475, [614] := 7291.35, [615] := 7303.225, [616] := 7315.1, [617] := 7326.975, [618] := 7338.85, [619] := 7350.725, [620] := 7362.6, [621] := 7374.475, [622] := 7386.35, [623] := 7398.225, [624] := 7410.1, [625] := 7421.975, [626] := 7433.85, [627] := 7445.725, [628] := 7457.6, [629] := 7469.475, [630] := 7481.35, [631] := 7493.225, [632] := 7505.1, [633] := 7516.975, [634] := 7528.85, [635] := 7540.725, [636] := 7552.6, [637] := 7564.475, [638] := 7576.35, [639] := 7588.225, [640] := 7600.1, [641] := 7611.975, [642] := 7623.85, [643] := 7635.725, [644] := 7647.6, [645] := 7659.475, [646] := 7671.35, [647] := 7683.225, [648] := 7695.1, [649] := 7706.975, [650] := 7718.85, [651] := 7730.725, [652] := 7742.6, [653] := 7754.475, [654] := 7766.35, [655] := 7778.225, [656] := 7790.1, [657] := 7801.975, [658] := 7813.85, [659] := 7825.725,
        [660] := 7837.6, [661] := 7849.475, [662] := 7861.35, [663] := 7873.225, [664] := 7885.1, [665] := 7896.975, [666] := 7908.85, [667] := 7920.725, [668] := 7932.6, [669] := 7944.475, [670] := 7956.35, [671] := 7968.225, [672] := 7980.1, [673] := 7991.975, [674] := 8003.85, [675] := 8015.725, [676] := 8027.6, [677] := 8039.475, [678] := 8051.35, [679] := 8063.225, [680] := 8075.1, [681] := 8086.975, [682] := 8098.85, [683] := 8110.725, [684] := 8122.6, [685] := 8134.475, [686] := 8146.35, [687] := 8158.225, [688] := 8170.1, [689] := 8181.975, [690] := 8193.85, [691] := 8205.725, [692] := 8217.6, [693] := 8229.475, [694] := 8241.35, [695] := 8253.225, [696] := 8265.1, [697] := 8276.975, [698] := 8288.85, [699] := 8300.725, [700] := 8312.6, [701] := 8324.475, [702] := 8336.35, [703] := 8348.225, [704] := 8360.1, [705] := 8371.975, [706] := 8383.85, [707] := 8395.725, [708] := 8407.6, [709] := 8419.475, [710] := 8431.35, [711] := 8443.225, [712] := 8455.1, [713] := 8466.975, [714] := 8478.85, [715] := 8490.725, [716] := 8502.6, [717] := 8514.475, [718] := 8526.35, [719] := 8538.225,
        [720] := 8550.1, [721] := 8561.975, [722] := 8573.85, [723] := 8585.725, [724] := 8597.6, [725] := 8609.475, [726] := 8621.35, [727] := 8633.225, [728] := 8645.1, [729] := 8656.975, [730] := 8668.85, [731] := 8680.725, [732] := 8692.6, [733] := 8704.475, [734] := 8716.35, [735] := 8728.225, [736] := 8740.1, [737] := 8751.975, [738] := 8763.85, [739] := 8775.725, [740] := 8787.6, [741] := 8799.475, [742] := 8811.35, [743] := 8823.225, [744] := 8835.1, [745] := 8846.975, [746] := 8858.85, [747] := 8870.725, [748] := 8882.6, [749] := 8894.475, [750] := 8906.35, [751] := 8918.225, [752] := 8930.1, [753] := 8941.975, [754] := 8953.85, [755] := 8965.725, [756] := 8977.6, [757] := 8989.475, [758] := 9001.35, [759] := 9013.225, [760] := 9025.1, [761] := 9036.975, [762] := 9048.85, [763] := 9060.725, [764] := 9072.6, [765] := 9084.475, [766] := 9096.35, [767] := 9108.225, [768] := 9120.1, [769] := 9131.975, [770] := 9143.85, [771] := 9155.725, [772] := 9167.6, [773] := 9179.475, [774] := 9191.35, [775] := 9203.225, [776] := 9215.1, [777] := 9226.975, [778] := 9238.85, [779] := 9250.725,
        [780] := 9262.6, [781] := 9274.475, [782] := 9286.35, [783] := 9298.225, [784] := 9310.1, [785] := 9321.975, [786] := 9333.85, [787] := 9345.725, [788] := 9357.6, [789] := 9369.475, [790] := 9381.35, [791] := 9393.225, [792] := 9405.1, [793] := 9416.975, [794] := 9428.85, [795] := 9440.725, [796] := 9452.6, [797] := 9464.475, [798] := 9476.35, [799] := 9499.9);
   QOP_HMI_GRAPH1_LINE1_DATAY : REAL[800] := ([0] := 8.640478, [1] := 12.048587, [2] := 16.15492, [3] := 11.545239, [4] := 12.803529, [5] := 13.150183, [6] := 16.406704, [7] := 18.917933, [8] := 18.303373, [9] := 14.9034, [10] := 14.452511, [11] := 16.967709, [12] := 17.523865, [13] := 17.528265, [14] := 15.852798, [15] := 19.847738, [16] := 21.58462, [17] := 20.698774, [18] := 19.38609, [19] := 18.922352, [20] := 19.0659, [21] := 23.344717, [22] := 25.906706, [23] := 22.89028, [24] := 22.01614, [25] := 19.309008, [26] := 22.309874, [27] := 24.439966, [28] := 23.178478, [29] := 19.866764, [30] := 20.686321, [31] := 23.127478, [32] := 26.317764, [33] := 25.30971, [34] := 20.165222, [35] := 20.417866, [36] := 21.856522, [37] := 25.094206, [38] := 23.377897, [39] := 22.370955, [40] := 23.175394, [41] := 23.494308, [42] := 23.194908, [43] := 25.065815, [44] := 24.964626, [45] := 25.241148, [46] := 24.267918, [47] := 25.40121, [48] := 25.486252, [49] := 22.381895, [50] := 24.748182, [51] := 23.032167, [52] := 25.833559, [53] := 24.900312, [54] := 22.731266, [55] := 24.602678, [56] := 23.31761, [57] := 23.34358, [58] := 28.173939, [59] := 25.401917,
        [60] := 27.500364, [61] := 26.71452, [62] := 30.053297, [63] := 24.665148, [64] := 28.382927, [65] := 25.512245, [66] := 26.476107, [67] := 26.147812, [68] := 25.636137, [69] := 24.800014, [70] := 27.736267, [71] := 25.578403, [72] := 27.738604, [73] := 23.771915, [74] := 20.071796, [75] := 20.436829, [76] := 24.933144, [77] := 23.683805, [78] := 22.84919, [79] := 20.665646, [80] := 20.731936, [81] := 21.633072, [82] := 23.324392, [83] := 23.903866, [84] := 21.74971, [85] := 22.815102, [86] := 24.04171, [87] := 27.229536, [88] := 23.471058, [89] := 21.558872, [90] := 23.144806, [91] := 23.722237, [92] := 25.48089, [93] := 23.050255, [94] := 22.624762, [95] := 23.149204, [96] := 22.278223, [97] := 25.079906, [98] := 24.208017, [99] := 21.5668, [100] := 21.891243, [101] := 22.996447, [102] := 25.097317, [103] := 25.236776, [104] := 23.311493, [105] := 17.522165, [106] := 18.220757, [107] := 20.978863, [108] := 23.043438, [109] := 18.218222, [110] := 17.937801, [111] := 19.80259, [112] := 25.465637, [113] := 22.0018, [114] := 21.272945, [115] := 18.929247, [116] := 18.960272, [117] := 23.8818, [118] := 25.50469, [119] := 19.973616,
        [120] := 21.636667, [121] := 19.010132, [122] := 24.228188, [123] := 28.241718, [124] := 21.604437, [125] := 21.715107, [126] := 20.99141, [127] := 22.643549, [128] := 25.281889, [129] := 22.556465, [130] := 22.507948, [131] := 20.802643, [132] := 20.503784, [133] := 25.909775, [134] := 23.414377, [135] := 18.744244, [136] := 20.150925, [137] := 22.552769, [138] := 24.009459, [139] := 23.276924, [140] := 19.480764, [141] := 20.932194, [142] := 22.39446, [143] := 21.863403, [144] := 23.009321, [145] := 20.029192, [146] := 19.780973, [147] := 20.91805, [148] := 22.238428, [149] := 21.062323, [150] := 19.037777, [151] := 17.814354, [152] := 19.85654, [153] := 18.29818, [154] := 20.202778, [155] := 13.840115, [156] := 16.030268, [157] := 17.098085, [158] := 18.559952, [159] := 17.630953, [160] := 17.37356, [161] := 19.249826, [162] := 18.785769, [163] := 18.975897, [164] := 17.403074, [165] := 14.322199, [166] := 19.204453, [167] := 19.509253, [168] := 18.461702, [169] := 22.771814, [170] := 18.067604, [171] := 16.220417, [172] := 18.948776, [173] := 20.116512, [174] := 20.123737, [175] := 16.300148, [176] := 16.346048, [177] := 18.735132, [178] := 22.160917, [179] := 20.738415,
        [180] := 15.011549, [181] := 14.870763, [182] := 17.061428, [183] := 18.61948, [184] := 16.50043, [185] := 14.061503, [186] := 16.229376, [187] := 14.010373, [188] := 21.169994, [189] := 18.333473, [190] := 14.413399, [191] := 13.386299, [192] := 16.839153, [193] := 15.991238, [194] := 18.60647, [195] := 14.80574, [196] := 12.712013, [197] := 16.13887, [198] := 16.666893, [199] := 20.77825, [200] := 11.967078, [201] := 15.008445, [202] := 9.917587, [203] := 18.353775, [204] := 20.055397, [205] := 19.311312, [206] := 14.870444, [207] := 15.52772, [208] := 24.185966, [209] := 18.68528, [210] := 20.503345, [211] := 16.261333, [212] := 18.064804, [213] := 18.130087, [214] := 22.85758, [215] := 19.969095, [216] := 17.74716, [217] := 16.358616, [218] := 22.128332, [219] := 17.930681, [220] := 18.670786, [221] := 15.162657, [222] := 15.947306, [223] := 17.423958, [224] := 19.888466, [225] := 15.391287, [226] := 15.118713, [227] := 14.714317, [228] := 12.673299, [229] := 17.082436, [230] := 13.129913, [231] := 11.013548, [232] := 13.414097, [233] := 13.18877, [234] := 16.901272, [235] := 15.590264, [236] := 13.453439, [237] := 12.266618, [238] := 14.338328, [239] := 16.596315,
        [240] := 14.410278, [241] := 14.268788, [242] := 12.808071, [243] := 15.726207, [244] := 16.398216, [245] := 16.326368, [246] := 11.720727, [247] := 15.365087, [248] := 14.073557, [249] := 17.015888, [250] := 13.404648, [251] := 13.253164, [252] := 13.153362, [253] := 14.013797, [254] := 16.096373, [255] := 14.048129, [256] := 10.200221, [257] := 12.5478325, [258] := 13.006595, [259] := 13.689388, [260] := 13.393411, [261] := 11.1881275, [262] := 10.457897, [263] := 14.905193, [264] := 15.718977, [265] := 13.104463, [266] := 12.147091, [267] := 12.3296585, [268] := 12.946945, [269] := 14.896856, [270] := 16.534145, [271] := 14.3876095, [272] := 12.354283, [273] := 14.621443, [274] := 15.901223, [275] := 16.571314, [276] := 14.068442, [277] := 19.430998, [278] := 17.792337, [279] := 21.411657, [280] := 16.630415, [281] := 17.52582, [282] := 17.496061, [283] := 18.107431, [284] := 21.260475, [285] := 17.455685, [286] := 18.419106, [287] := 16.268911, [288] := 22.103226, [289] := 20.27059, [290] := 21.56848, [291] := 16.873173, [292] := 16.056686, [293] := 14.460966, [294] := 18.967585, [295] := 15.762669, [296] := 18.021883, [297] := 14.186476, [298] := 18.324547, [299] := 18.214905,
        [300] := 19.621658, [301] := 15.70497, [302] := 15.298011, [303] := 14.559314, [304] := 18.993305, [305] := 18.458313, [306] := 16.693691, [307] := 13.7706175, [308] := 15.30108, [309] := 15.574576, [310] := 18.284393, [311] := 15.299471, [312] := 15.329131, [313] := 13.026953, [314] := 18.204666, [315] := 15.515316, [316] := 15.8075075, [317] := 12.359796, [318] := 15.062981, [319] := 14.066408, [320] := 17.63001, [321] := 15.786794, [322] := 13.918246, [323] := 13.523747, [324] := 16.382256, [325] := 14.816695, [326] := 15.618403, [327] := 14.626831, [328] := 13.211405, [329] := 13.628054, [330] := 17.303356, [331] := 15.178338, [332] := 14.172891, [333] := 13.589308, [334] := 16.918009, [335] := 14.528158, [336] := 14.956, [337] := 12.394834, [338] := 14.495136, [339] := 15.88853, [340] := 15.831939, [341] := 17.080986, [342] := 14.996176, [343] := 16.863619, [344] := 15.341717, [345] := 20.318169, [346] := 16.011501, [347] := 14.290029, [348] := 14.4714985, [349] := 16.914492, [350] := 15.8386965, [351] := 15.78798, [352] := 15.799642, [353] := 16.465462, [354] := 15.521789, [355] := 20.236143, [356] := 17.902172, [357] := 16.212862, [358] := 13.067386, [359] := 16.51617,
        [360] := 17.175379, [361] := 16.72182, [362] := 14.523548, [363] := 16.153185, [364] := 15.868513, [365] := 21.303112, [366] := 14.433191, [367] := 14.616021, [368] := 11.455869, [369] := 18.21042, [370] := 16.107609, [371] := 19.351856, [372] := 15.087788, [373] := 14.24472, [374] := 14.197935, [375] := 16.466179, [376] := 16.25453, [377] := 13.69018, [378] := 13.396828, [379] := 14.496634, [380] := 16.497238, [381] := 17.05558, [382] := 14.441198, [383] := 12.314985, [384] := 13.345281, [385] := 14.702249, [386] := 16.187485, [387] := 13.208093, [388] := 12.337284, [389] := 13.144382, [390] := 15.40766, [391] := 18.534473, [392] := 14.352261, [393] := 9.959378, [394] := 11.023494, [395] := 12.720478, [396] := 15.262413, [397] := 11.530024, [398] := 11.665546, [399] := 10.9605465, [400] := 13.901475, [401] := 16.364332, [402] := 12.513104, [403] := 9.630932, [404] := 10.101231, [405] := 13.051876, [406] := 14.948949, [407] := 14.391801, [408] := 11.760865, [409] := 11.50673, [410] := 17.496887, [411] := 15.809467, [412] := 15.003649, [413] := 14.490398, [414] := 12.892191, [415] := 14.387138, [416] := 20.087578, [417] := 17.07833, [418] := 15.865026, [419] := 13.827329,
        [420] := 19.659092, [421] := 18.156387, [422] := 15.823868, [423] := 14.324835, [424] := 16.30502, [425] := 17.66098, [426] := 18.329336, [427] := 16.740936, [428] := 13.446152, [429] := 14.914333, [430] := 16.391006, [431] := 17.78955, [432] := 16.551067, [433] := 13.447825, [434] := 14.474585, [435] := 15.54957, [436] := 17.89549, [437] := 16.663305, [438] := 16.778881, [439] := 15.052992, [440] := 17.406229, [441] := 16.10572, [442] := 15.501981, [443] := 14.668393, [444] := 13.9603405, [445] := 16.886969, [446] := 16.74086, [447] := 16.87651, [448] := 12.642175, [449] := 15.50693, [450] := 14.47079, [451] := 17.203062, [452] := 15.805708, [453] := 13.43635, [454] := 12.973783, [455] := 13.396793, [456] := 15.792852, [457] := 16.563019, [458] := 11.326519, [459] := 12.7078085, [460] := 12.421941, [461] := 14.513323, [462] := 12.465783, [463] := 11.881115, [464] := 11.29337, [465] := 14.120512, [466] := 16.200369, [467] := 16.986618, [468] := 10.129402, [469] := 13.250645, [470] := 12.101928, [471] := 15.890871, [472] := 13.496785, [473] := 14.268001, [474] := 10.844959, [475] := 15.116546, [476] := 17.261196, [477] := 18.72781, [478] := 14.270488, [479] := 16.13396,
        [480] := 13.175228, [481] := 20.924582, [482] := 18.935307, [483] := 19.895336, [484] := 19.42641, [485] := 20.823307, [486] := 20.464397, [487] := 21.745216, [488] := 19.400858, [489] := 17.278854, [490] := 20.43975, [491] := 21.182156, [492] := 23.640287, [493] := 22.633343, [494] := 18.515873, [495] := 18.65536, [496] := 19.013926, [497] := 18.796803, [498] := 17.271997, [499] := 16.739592, [500] := 17.214983, [501] := 18.823338, [502] := 19.769547, [503] := 18.22185, [504] := 14.417278, [505] := 14.833816, [506] := 15.032705, [507] := 18.85127, [508] := 17.376423, [509] := 13.468308, [510] := 12.922536, [511] := 16.828295, [512] := 17.677944, [513] := 15.166903, [514] := 12.757465, [515] := 12.295368, [516] := 14.171704, [517] := 17.705408, [518] := 15.417311, [519] := 13.343057, [520] := 14.2880335, [521] := 16.19597, [522] := 18.201586, [523] := 14.751246, [524] := 14.992276, [525] := 10.61734, [526] := 15.644738, [527] := 16.784288, [528] := 18.833946, [529] := 13.720218, [530] := 15.42867, [531] := 13.870568, [532] := 17.58353, [533] := 14.311899, [534] := 13.667319, [535] := 11.960621, [536] := 15.271391, [537] := 17.122808, [538] := 15.213961, [539] := 12.10625,
        [540] := 14.424803, [541] := 12.544974, [542] := 17.04722, [543] := 13.438442, [544] := 15.522103, [545] := 13.861137, [546] := 14.436155, [547] := 17.972378, [548] := 14.085312, [549] := 14.698985, [550] := 14.601633, [551] := 14.555192, [552] := 17.719355, [553] := 15.505059, [554] := 14.66584, [555] := 15.869474, [556] := 16.73342, [557] := 17.399458, [558] := 14.4624815, [559] := 15.504263, [560] := 15.329877, [561] := 17.440504, [562] := 19.353046, [563] := 18.67909, [564] := 15.744633, [565] := 17.28334, [566] := 15.943556, [567] := 22.21156, [568] := 15.539855, [569] := 16.65994, [570] := 14.81744, [571] := 16.897034, [572] := 16.445004, [573] := 19.334883, [574] := 13.806719, [575] := 15.5185995, [576] := 13.349025, [577] := 17.88267, [578] := 17.124548, [579] := 15.508641, [580] := 12.358196, [581] := 15.661362, [582] := 11.897347, [583] := 15.704539, [584] := 13.283918, [585] := 11.877828, [586] := 9.954816, [587] := 15.60111, [588] := 13.407782, [589] := 12.879649, [590] := 9.236331, [591] := 10.159274, [592] := 15.711695, [593] := 15.362379, [594] := 10.968168, [595] := 7.027807, [596] := 8.941284, [597] := 10.2645855, [598] := 12.419368, [599] := 8.142633,
        [600] := 9.935912, [601] := 6.811412, [602] := 12.204977, [603] := 12.430342, [604] := 11.413118, [605] := 7.634844, [606] := 7.3944674, [607] := 10.941769, [608] := 11.819309, [609] := 10.945043, [610] := 6.3290224, [611] := 9.430959, [612] := 9.970676, [613] := 13.957617, [614] := 12.324294, [615] := 9.511663, [616] := 7.328467, [617] := 11.078566, [618] := 14.117945, [619] := 10.395471, [620] := 12.460189, [621] := 11.970919, [622] := 11.1806, [623] := 15.382232, [624] := 11.643698, [625] := 13.042871, [626] := 12.909826, [627] := 11.836311, [628] := 15.371323, [629] := 13.572518, [630] := 11.734415, [631] := 12.120197, [632] := 11.11358, [633] := 15.995571, [634] := 12.399776, [635] := 12.930518, [636] := 13.135661, [637] := 13.8306465, [638] := 15.817931, [639] := 11.411335, [640] := 9.975585, [641] := 11.27249, [642] := 10.611791, [643] := 13.859974, [644] := 11.292364, [645] := 10.673416, [646] := 11.972852, [647] := 12.0122385, [648] := 14.363191, [649] := 11.7645855, [650] := 7.6808496, [651] := 8.101966, [652] := 9.766522, [653] := 9.343901, [654] := 7.7460847, [655] := 9.427936, [656] := 7.914462, [657] := 9.472275, [658] := 12.530629, [659] := 10.122815,
        [660] := 5.4975214, [661] := 5.5360966, [662] := 8.111877, [663] := 10.21814, [664] := 8.623204, [665] := 7.1391573, [666] := 4.1548533, [667] := 4.862055, [668] := 7.113561, [669] := 11.962316, [670] := 6.201153, [671] := 5.862428, [672] := 9.188898, [673] := 9.34941, [674] := 7.1172, [675] := 5.169464, [676] := 5.421927, [677] := 6.049053, [678] := 4.2964516, [679] := 10.6102085, [680] := 8.139837, [681] := 7.354653, [682] := 6.1096573, [683] := 9.007132, [684] := 10.052336, [685] := 7.214447, [686] := 11.142412, [687] := 11.616147, [688] := 12.898207, [689] := 13.986545, [690] := 10.940733, [691] := 11.178188, [692] := 13.443853, [693] := 14.440242, [694] := 14.413773, [695] := 11.29955, [696] := 8.455722, [697] := 8.052245, [698] := 11.634937, [699] := 12.031427, [700] := 9.679282, [701] := 6.7846274, [702] := 5.729657, [703] := 7.282798, [704] := 10.9099455, [705] := 9.089022, [706] := 8.593963, [707] := 6.01949, [708] := 7.44693, [709] := 9.48813, [710] := 7.8323565, [711] := 6.875585, [712] := 3.5279686, [713] := 5.783084, [714] := 7.365003, [715] := 5.9141717, [716] := 3.553874, [717] := 3.235494, [718] := 6.940142, [719] := 6.268097,
        [720] := 4.5149336, [721] := 2.727029, [722] := 2.858635, [723] := 1.6195867, [724] := 4.288746, [725] := 4.213401, [726] := 2.3946638, [727] := 1.3257987, [728] := 2.9358242, [729] := 3.941673, [730] := 1.0061519, [731] := 1.4037433, [732] := 1.8825223, [733] := 2.9126854, [734] := 1.9244548, [735] := 1.3394253, [736] := 2.7016873, [737] := 0.81737137, [738] := 3.3105254, [739] := 3.3060334, [740] := 2.4629314, [741] := 1.6427113, [742] := 2.1391842, [743] := 1.8267757, [744] := 5.549308, [745] := 1.3398166, [746] := 0.5171795, [747] := 3.5485892, [748] := 3.8085148, [749] := 3.9093091, [750] := 2.5730128, [751] := 3.8541727, [752] := 2.9804597, [753] := 5.930102, [754] := 7.0776677, [755] := 4.488744, [756] := 2.748872, [757] := 3.5492651, [758] := 2.9792347, [759] := 1.5129887, [760] := 0.38204575, [761] := 0.44168258, [762] := 3.469824, [763] := 4.0030203, [764] := 1.5054841, [765] := 0.36415577, [766] := 1.1133915, [767] := 4.2726665, [768] := 1.4018575, [769] := 1.6086522, [770] := 2.9790049, [771] := 0.14037865, [772] := 2.8836489, [773] := 1.4167106, [774] := 4.495777, [775] := 5.2685127, [776] := 0.8242176, [777] := 0.24358825, [778] := 1.0160031, [779] := 1.9442765,
        [780] := 2.7556272, [781] := 0.9068259, [782] := 1.5153481, [783] := 0.6783843, [784] := 3.564265, [785] := 2.5476072, [786] := 2.005307, [787] := 1.4849061, [788] := 3.627693, [789] := 2.6940117, [790] := 1.0323902, [791] := 1.2012544, [792] := 3.5953825, [793] := 2.329525, [794] := 3.4884062, [795] := 3.4473772, [796] := 2.9199097, [797] := 1.9954675, [798] := 0.25379607);
   QOP_HMI_GRAPH1_LINE1_HDR : REAL[10] := ([0] := 800.0, [4] := 40.0);
        [3]   // Hide line
        [0]   // Samples
        [4]   // Updater
        [5]   // Pointer
   QOP_HMI_GRAPH1_LINE2_DATAY : REAL[800] := ([1] := 3.3534036, [2] := 3.531193, [3] := 6.9746075, [4] := 6.637278, [5] := 3.612531, [6] := 3.6597059, [7] := 0.6001284, [8] := 1.7796569, [9] := 4.3503356, [10] := 2.691565, [11] := 0.19508517, [12] := 0.26164955, [13] := 2.5085707, [14] := 3.0051093, [15] := 5.4986057, [16] := 0.697083, [17] := 0.033587493, [18] := 2.463493, [19] := 4.0523, [20] := 7.2753863, [21] := 3.0235496, [22] := 1.0354353, [23] := 1.3047848, [24] := 1.3198193, [25] := 2.8475754, [26] := 1.1883657, [27] := 4.1902227, [28] := 2.2279334, [29] := 0.788623, [30] := 0.99260455, [31] := 0.401114, [32] := 4.6000314, [33] := 2.5748675, [34] := 1.3914604, [35] := 2.8033254, [36] := 3.745095, [37] := 0.3081683, [38] := 0.8623208, [39] := 1.4603868, [40] := 1.974174, [41] := 1.0342271, [42] := 0.137183, [43] := 1.0590727, [44] := 0.38672403, [45] := 2.086014, [46] := 2.6104805, [47] := 1.9002116, [48] := 0.86431277, [49] := 1.4920416, [50] := 0.81076443, [51] := 1.8687118, [52] := 2.041205, [53] := 4.65186, [54] := 4.6413713, [55] := 6.1021237, [56] := 7.4492207, [57] := 1.7641082, [58] := 1.9688655, [59] := 2.699051, [60] := 1.1358045,
        [61] := 2.9261239, [62] := 2.3378615, [63] := 1.7159932, [64] := 1.7102897, [65] := 0.6254604, [66] := 0.5693241, [67] := 2.0473926, [68] := 2.5646367, [69] := 0.3251939, [70] := 0.7480395, [71] := 0.8355189, [72] := 2.4415507, [73] := 3.591917, [74] := 0.37543106, [75] := 0.005546573, [76] := 2.8007097, [77] := 1.2996446, [78] := 1.8856496, [79] := 2.9974678, [80] := 3.6525474, [81] := 4.097563, [82] := 2.5882862, [83] := 6.6334543, [84] := 6.0551414, [85] := 3.9450135, [86] := 4.725222, [87] := 2.3244197, [88] := 2.3760698, [89] := 4.680808, [90] := 4.796606, [91] := 7.5569735, [92] := 4.312654, [93] := 3.2010977, [94] := 6.424852, [95] := 7.412713, [96] := 4.502274, [97] := 1.589109, [98] := 0.49255145, [99] := 3.2436614, [100] := 4.3194194, [101] := 5.896507, [102] := 2.54729, [103] := 3.4243033, [104] := 5.0324807, [105] := 6.798377, [106] := 6.5803194, [107] := 6.362151, [108] := 3.0292168, [109] := 3.935463, [110] := 7.2975883, [111] := 10.926903, [112] := 8.63196, [113] := 7.1426573, [114] := 8.015392, [115] := 9.259606, [116] := 8.470437, [117] := 4.971822, [118] := 8.002744, [119] := 9.048179, [120] := 9.75717,
        [121] := 9.055082, [122] := 4.995378, [123] := 5.1977744, [124] := 2.641848, [125] := 5.4031224, [126] := 6.9232554, [127] := 6.8322287, [128] := 1.4356799, [129] := 6.035524, [130] := 6.4531775, [131] := 8.507023, [132] := 5.482772, [133] := 3.5633225, [134] := 3.2568421, [135] := 4.082192, [136] := 8.964332, [137] := 4.4167376, [138] := 3.262563, [139] := 5.9650207, [140] := 7.2031164, [141] := 7.0080085, [142] := 5.946525, [143] := 5.4425178, [144] := 5.826893, [145] := 9.182988, [146] := 9.969742, [147] := 10.94666, [148] := 6.748839, [149] := 7.849214, [150] := 8.574109, [151] := 9.924865, [152] := 9.404089, [153] := 4.6317606, [154] := 8.167865, [155] := 10.725103, [156] := 11.455436, [157] := 14.379229, [158] := 7.5518713, [159] := 9.869151, [160] := 13.029636, [161] := 9.2464, [162] := 13.900441, [163] := 11.097954, [164] := 12.782827, [165] := 13.948518, [166] := 14.484993, [167] := 14.422527, [168] := 10.967426, [169] := 13.456744, [170] := 13.043097, [171] := 13.3050785, [172] := 13.264954, [173] := 11.305839, [174] := 13.436386, [175] := 15.378491, [176] := 12.78722, [177] := 13.590341, [178] := 8.408154, [179] := 10.842074, [180] := 13.378816,
        [181] := 14.97371, [182] := 14.643065, [183] := 9.855993, [184] := 12.530187, [185] := 14.545814, [186] := 14.132418, [187] := 13.641665, [188] := 10.309085, [189] := 11.037568, [190] := 10.684323, [191] := 14.892991, [192] := 13.853296, [193] := 8.331038, [194] := 11.261816, [195] := 13.756248, [196] := 15.081258, [197] := 12.364619, [198] := 12.832242, [199] := 9.838357, [200] := 13.030633, [201] := 13.949508, [202] := 17.126354, [203] := 11.453867, [204] := 12.828083, [205] := 12.24678, [206] := 16.102608, [207] := 14.792684, [208] := 14.290717, [209] := 11.630066, [210] := 13.823835, [211] := 15.691286, [212] := 16.84324, [213] := 13.173003, [214] := 11.054565, [215] := 10.444025, [216] := 13.280423, [217] := 15.33694, [218] := 10.835184, [219] := 13.614946, [220] := 11.110012, [221] := 15.345936, [222] := 14.226459, [223] := 13.93595, [224] := 10.053516, [225] := 14.650016, [226] := 13.175689, [227] := 16.101572, [228] := 12.951012, [229] := 15.736699, [230] := 13.361854, [231] := 16.485905, [232] := 14.47832, [233] := 16.71535, [234] := 12.17504, [235] := 13.935441, [236] := 13.683197, [237] := 17.723778, [238] := 17.38144, [239] := 13.160875, [240] := 13.118609,
        [241] := 16.861647, [242] := 15.056183, [243] := 16.695892, [244] := 12.489058, [245] := 13.450212, [246] := 17.444784, [247] := 18.33834, [248] := 17.379843, [249] := 13.66699, [250] := 18.05315, [251] := 15.210706, [252] := 16.083115, [253] := 15.318972, [254] := 15.336999, [255] := 13.377054, [256] := 15.5930805, [257] := 17.653759, [258] := 16.749283, [259] := 11.834438, [260] := 12.598642, [261] := 15.750241, [262] := 17.288988, [263] := 13.184794, [264] := 11.638729, [265] := 8.81311, [266] := 14.389783, [267] := 14.081394, [268] := 12.017945, [269] := 7.4954085, [270] := 9.692651, [271] := 10.401228, [272] := 10.347632, [273] := 12.232635, [274] := 10.611756, [275] := 8.621272, [276] := 12.805931, [277] := 14.324129, [278] := 12.057029, [279] := 10.853888, [280] := 10.711576, [281] := 13.316401, [282] := 13.872786, [283] := 13.293834, [284] := 11.541196, [285] := 9.361029, [286] := 14.36809, [287] := 17.36042, [288] := 16.272774, [289] := 10.322908, [290] := 10.819645, [291] := 14.131609, [292] := 13.692302, [293] := 14.104554, [294] := 11.702457, [295] := 10.119688, [296] := 13.61416, [297] := 15.105926, [298] := 15.664339, [299] := 10.843025, [300] := 7.8441677,
        [301] := 11.06647, [302] := 14.951086, [303] := 17.240461, [304] := 10.740415, [305] := 10.174738, [306] := 13.456628, [307] := 16.295572, [308] := 14.944225, [309] := 10.739576, [310] := 9.390945, [311] := 10.956314, [312] := 14.195315, [313] := 16.071491, [314] := 12.2400675, [315] := 12.329349, [316] := 12.378265, [317] := 15.751298, [318] := 12.998554, [319] := 14.108398, [320] := 11.145385, [321] := 14.164908, [322] := 13.206734, [323] := 18.881023, [324] := 10.510352, [325] := 11.2263775, [326] := 11.477764, [327] := 15.320555, [328] := 14.110281, [329] := 16.434748, [330] := 11.433756, [331] := 11.923144, [332] := 15.707338, [333] := 14.994532, [334] := 10.614503, [335] := 11.262534, [336] := 10.774004, [337] := 12.916483, [338] := 12.625863, [339] := 14.078, [340] := 13.0792055, [341] := 13.74429, [342] := 12.400012, [343] := 16.241163, [344] := 12.853171, [345] := 11.1838, [346] := 9.471174, [347] := 13.8638735, [348] := 13.101122, [349] := 15.063375, [350] := 11.796584, [351] := 10.870054, [352] := 12.889628, [353] := 11.182414, [354] := 11.885725, [355] := 7.167679, [356] := 11.869752, [357] := 12.637882, [358] := 15.304512, [359] := 13.640565, [360] := 12.238953,
        [361] := 12.452256, [362] := 16.070183, [363] := 17.829443, [364] := 17.347054, [365] := 14.5624075, [366] := 13.474633, [367] := 16.613874, [368] := 19.01979, [369] := 16.796799, [370] := 14.507098, [371] := 13.312371, [372] := 18.742582, [373] := 16.596582, [374] := 17.767208, [375] := 14.064208, [376] := 13.908845, [377] := 16.14046, [378] := 17.133396, [379] := 17.123636, [380] := 16.763165, [381] := 13.273631, [382] := 16.68615, [383] := 18.298227, [384] := 18.959423, [385] := 14.962935, [386] := 13.032571, [387] := 14.779658, [388] := 19.914658, [389] := 16.107042, [390] := 15.680122, [391] := 10.742471, [392] := 15.264705, [393] := 13.896753, [394] := 17.80672, [395] := 10.781497, [396] := 13.762799, [397] := 13.980612, [398] := 15.383172, [399] := 14.41513, [400] := 16.151459, [401] := 10.045757, [402] := 14.319163, [403] := 20.035934, [404] := 17.035309, [405] := 16.320913, [406] := 12.5232115, [407] := 14.001896, [408] := 14.773104, [409] := 18.229195, [410] := 16.563358, [411] := 11.739884, [412] := 15.255901, [413] := 15.978071, [414] := 17.62166, [415] := 14.174024, [416] := 12.412751, [417] := 13.662979, [418] := 13.460283, [419] := 16.241835, [420] := 14.950174,
        [421] := 13.453403, [422] := 13.511281, [423] := 15.223826, [424] := 14.535408, [425] := 16.697023, [426] := 10.488997, [427] := 14.685702, [428] := 15.051703, [429] := 17.65663, [430] := 14.475721, [431] := 13.975298, [432] := 13.86466, [433] := 16.451668, [434] := 15.820405, [435] := 16.87704, [436] := 12.705734, [437] := 14.170586, [438] := 15.806153, [439] := 18.667274, [440] := 15.555671, [441] := 13.741625, [442] := 14.580885, [443] := 17.621706, [444] := 16.584301, [445] := 17.107132, [446] := 7.8874893, [447] := 16.561453, [448] := 12.942871, [449] := 17.895552, [450] := 15.000397, [451] := 12.553737, [452] := 14.207421, [453] := 17.47158, [454] := 14.000662, [455] := 15.13385, [456] := 13.014131, [457] := 14.31624, [458] := 16.79038, [459] := 16.673536, [460] := 17.201979, [461] := 12.203155, [462] := 14.151995, [463] := 14.970671, [464] := 16.363398, [465] := 15.641793, [466] := 12.588949, [467] := 12.990771, [468] := 14.430229, [469] := 13.846946, [470] := 14.429775, [471] := 10.114635, [472] := 9.611441, [473] := 11.1671505, [474] := 10.727707, [475] := 10.924264, [476] := 12.635943, [477] := 11.168024, [478] := 12.423691, [479] := 13.850453, [480] := 15.1602,
        [481] := 11.220139, [482] := 11.888793, [483] := 11.864083, [484] := 14.433583, [485] := 13.253095, [486] := 15.596853, [487] := 13.650823, [488] := 14.542465, [489] := 15.813312, [490] := 14.40857, [491] := 11.506729, [492] := 11.184566, [493] := 10.216492, [494] := 12.729207, [495] := 13.083607, [496] := 14.08557, [497] := 11.297289, [498] := 13.689083, [499] := 12.275739, [500] := 15.798857, [501] := 10.412629, [502] := 10.871239, [503] := 11.253646, [504] := 15.533872, [505] := 14.843425, [506] := 14.516912, [507] := 11.965866, [508] := 12.691516, [509] := 14.99366, [510] := 17.27663, [511] := 13.274494, [512] := 12.623464, [513] := 13.959466, [514] := 14.245865, [515] := 17.492048, [516] := 14.715765, [517] := 13.017315, [518] := 12.897484, [519] := 14.598769, [520] := 15.653661, [521] := 14.386821, [522] := 14.557609, [523] := 14.098562, [524] := 16.849426, [525] := 17.315874, [526] := 15.053304, [527] := 13.0019, [528] := 12.510368, [529] := 15.507197, [530] := 14.284923, [531] := 13.364887, [532] := 9.804605, [533] := 12.200399, [534] := 12.938601, [535] := 13.507409, [536] := 13.274283, [537] := 11.914207, [538] := 11.406046, [539] := 13.795453, [540] := 10.587915,
        [541] := 16.295187, [542] := 9.944294, [543] := 12.832883, [544] := 13.344577, [545] := 14.336258, [546] := 12.990956, [547] := 12.390576, [548] := 12.182315, [549] := 14.110604, [550] := 14.688033, [551] := 14.585722, [552] := 10.734396, [553] := 13.049343, [554] := 13.573705, [555] := 16.28553, [556] := 13.641591, [557] := 9.927377, [558] := 9.580294, [559] := 15.95495, [560] := 15.22545, [561] := 15.913257, [562] := 12.337992, [563] := 13.663665, [564] := 16.559765, [565] := 17.753326, [566] := 17.271542, [567] := 9.766834, [568] := 11.25086, [569] := 17.015778, [570] := 17.881584, [571] := 16.152176, [572] := 14.936061, [573] := 14.978764, [574] := 18.196787, [575] := 17.941618, [576] := 16.631645, [577] := 14.799148, [578] := 15.04164, [579] := 17.837723, [580] := 19.518883, [581] := 17.83391, [582] := 16.839783, [583] := 12.363979, [584] := 17.61389, [585] := 15.973538, [586] := 18.685188, [587] := 15.921065, [588] := 16.223036, [589] := 16.2894, [590] := 17.201069, [591] := 17.781544, [592] := 19.130302, [593] := 16.046736, [594] := 18.216663, [595] := 20.68556, [596] := 20.292767, [597] := 18.588446, [598] := 18.122347, [599] := 15.803492, [600] := 19.123922,
        [601] := 21.000061, [602] := 16.140282, [603] := 18.812965, [604] := 16.222174, [605] := 21.034826, [606] := 21.146614, [607] := 22.696203, [608] := 16.29868, [609] := 17.032883, [610] := 21.32483, [611] := 21.547136, [612] := 20.312862, [613] := 19.058067, [614] := 16.050198, [615] := 17.459639, [616] := 19.723633, [617] := 19.29277, [618] := 13.021853, [619] := 15.937635, [620] := 16.97579, [621] := 19.958998, [622] := 17.046106, [623] := 16.807981, [624] := 19.890448, [625] := 19.43576, [626] := 22.030132, [627] := 19.12567, [628] := 16.899284, [629] := 16.698212, [630] := 18.2982, [631] := 23.750921, [632] := 19.164877, [633] := 16.383162, [634] := 20.64179, [635] := 18.830927, [636] := 21.558966, [637] := 19.24943, [638] := 15.551351, [639] := 17.328115, [640] := 17.260323, [641] := 21.154066, [642] := 19.0468, [643] := 13.878459, [644] := 17.136967, [645] := 19.135414, [646] := 20.180828, [647] := 17.682808, [648] := 13.697943, [649] := 15.739703, [650] := 19.285921, [651] := 18.37105, [652] := 16.888206, [653] := 15.231101, [654] := 16.0276, [655] := 20.339218, [656] := 20.903152, [657] := 17.67488, [658] := 16.02597, [659] := 19.161158, [660] := 23.17093,
        [661] := 20.360617, [662] := 22.726202, [663] := 18.937353, [664] := 18.247414, [665] := 21.246302, [666] := 21.18673, [667] := 19.699678, [668] := 13.690877, [669] := 18.114685, [670] := 22.236523, [671] := 20.106363, [672] := 20.462288, [673] := 14.250034, [674] := 17.939167, [675] := 15.461999, [676] := 17.880611, [677] := 21.612003, [678] := 16.925789, [679] := 12.489276, [680] := 14.669352, [681] := 20.067245, [682] := 22.076044, [683] := 17.296345, [684] := 15.587112, [685] := 16.223154, [686] := 18.250462, [687] := 19.36003, [688] := 19.834713, [689] := 16.3245, [690] := 19.251633, [691] := 20.260218, [692] := 20.819197, [693] := 18.235989, [694] := 17.732533, [695] := 18.923775, [696] := 19.047169, [697] := 21.735662, [698] := 19.71062, [699] := 18.580208, [700] := 19.036346, [701] := 21.5035, [702] := 21.2059, [703] := 21.207132, [704] := 15.48786, [705] := 19.550436, [706] := 20.620295, [707] := 22.33095, [708] := 22.210495, [709] := 20.545181, [710] := 19.200497, [711] := 19.513308, [712] := 21.4225, [713] := 19.100145, [714] := 16.988844, [715] := 19.64293, [716] := 19.9873, [717] := 21.588472, [718] := 19.970598, [719] := 14.409454, [720] := 17.383928,
        [721] := 19.327412, [722] := 20.565762, [723] := 20.777685, [724] := 16.805939, [725] := 18.528303, [726] := 19.37562, [727] := 21.735697, [728] := 20.073841, [729] := 19.247503, [730] := 20.02834, [731] := 19.041296, [732] := 20.380486, [733] := 22.116304, [734] := 17.668425, [735] := 21.277456, [736] := 22.595186, [737] := 24.246948, [738] := 23.149628, [739] := 17.357126, [740] := 21.476015, [741] := 22.71142, [742] := 26.04467, [743] := 21.988308, [744] := 21.479992, [745] := 24.526396, [746] := 23.549984, [747] := 23.510561, [748] := 24.071608, [749] := 17.624638, [750] := 19.939545, [751] := 22.556492, [752] := 23.858435, [753] := 21.978899, [754] := 20.932724, [755] := 19.849625, [756] := 24.096542, [757] := 23.63772, [758] := 21.157537, [759] := 19.49075, [760] := 17.366533, [761] := 22.858536, [762] := 24.420828, [763] := 23.876585, [764] := 18.861332, [765] := 18.378832, [766] := 21.68609, [767] := 22.549055, [768] := 22.326275, [769] := 20.646109, [770] := 18.127602, [771] := 18.47078, [772] := 24.41515, [773] := 21.711153, [774] := 17.97576, [775] := 18.38137, [776] := 19.574211, [777] := 22.230633, [778] := 21.16217, [779] := 18.963543, [780] := 16.409594,
        [781] := 18.660965, [782] := 21.435509, [783] := 19.68947, [784] := 17.640612, [785] := 13.542736, [786] := 14.150061, [787] := 17.458305, [788] := 17.349478, [789] := 17.332298, [790] := 16.46534, [791] := 17.662197, [792] := 17.953644, [793] := 17.154943, [794] := 13.318513, [795] := 9.91505, [796] := 12.099397, [797] := 13.8664665, [798] := 14.923033, [799] := 8.008025);
   QOP_HMI_GRAPH2_HDR : REAL[10] := ([4] := 1.0, [5] := 26.659199, [6] := 20.0, [7] := 1.0);
   QOP_HMI_GRAPH2_LINE1_DATAX : REAL[800] := ([0] := 0.1, [1] := 0.08, [2] := 0.06, [3] := 0.04, [4] := 0.02, [6] := -0.02, [7] := -0.04, [8] := -0.06, [9] := -0.08, [10] := -0.099999994, [11] := -0.11999999, [12] := -0.13999999, [13] := -0.15999998, [14] := -0.17999998, [15] := -0.19999997, [16] := -0.21999997, [17] := -0.23999996, [18] := -0.25999996, [19] := -0.27999997, [20] := -0.29999998, [21] := -0.32, [22] := -0.34, [23] := -0.36, [24] := -0.38000003, [25] := -0.40000004, [26] := -0.42000005, [27] := -0.44000006, [28] := -0.46000007, [29] := -0.48000008, [30] := -0.50000006, [31] := -0.52000004, [32] := -0.54, [33] := -0.56, [34] := -0.58, [35] := -0.59999996, [36] := -0.61999995, [37] := -0.6399999, [38] := -0.6599999, [39] := -0.6799999, [40] := -0.69999987, [41] := -0.71999985, [42] := -0.73999983, [43] := -0.7599998, [44] := -0.7799998, [45] := -0.7999998, [46] := -0.81999975, [47] := -0.83999974, [48] := -0.8599997, [49] := -0.8799997, [50] := -0.8999997, [51] := -0.91999966, [52] := -0.93999964, [53] := -0.9599996, [54] := -0.9799996, [55] := -0.9999996, [56] := -1.0199996, [57] := -1.0399996, [58] := -1.0599996, [59] := -1.0799996, [60] := -1.0999995,
        [61] := -1.1199995, [62] := -1.1399995, [63] := -1.1599995, [64] := -1.1799995, [65] := -1.1999995, [66] := -1.2199994, [67] := -1.2399994, [68] := -1.2599994, [69] := -1.2799994, [70] := -1.2999994, [71] := -1.3199993, [72] := -1.3399993, [73] := -1.3599993, [74] := -1.3799993, [75] := -1.3999993, [76] := -1.4199992, [77] := -1.4399992, [78] := -1.4599992, [79] := -1.4799992, [80] := -1.4999992, [81] := -1.5199991, [82] := -1.5399991, [83] := -1.5599991, [84] := -1.5799991, [85] := -1.5999991, [86] := -1.619999, [87] := -1.639999, [88] := -1.659999, [89] := -1.679999, [90] := -1.699999, [91] := -1.719999, [92] := -1.7399989, [93] := -1.7599989, [94] := -1.7799989, [95] := -1.7999989, [96] := -1.8199989, [97] := -1.8399988, [98] := -1.8599988, [99] := -1.8799988, [100] := -1.8999988, [101] := -1.9199988, [102] := -1.9399987, [103] := -1.9599987, [104] := -1.9799987, [105] := -1.9999987, [106] := -2.0199988, [107] := -2.0399988, [108] := -2.0599988, [109] := -2.0799987, [110] := -2.0999987, [111] := -2.1199987, [112] := -2.1399987, [113] := -2.1599987, [114] := -2.1799986, [115] := -2.1999986, [116] := -2.2199986, [117] := -2.2399986, [118] := -2.2599986, [119] := -2.2799985, [120] := -2.2999985,
        [121] := -2.3199985, [122] := -2.3399985, [123] := -2.3599985, [124] := -2.3799984, [125] := -2.3999984, [126] := -2.4199984, [127] := -2.4399984, [128] := -2.4599984, [129] := -2.4799984, [130] := -2.4999983, [131] := -2.5199983, [132] := -2.5399983, [133] := -2.5599983, [134] := -2.5799983, [135] := -2.5999982, [136] := -2.6199982, [137] := -2.6399982, [138] := -2.6599982, [139] := -2.6799982, [140] := -2.6999981, [141] := -2.7199981, [142] := -2.739998, [143] := -2.759998, [144] := -2.779998, [145] := -2.799998, [146] := -2.819998, [147] := -2.839998, [148] := -2.859998, [149] := -2.879998, [150] := -2.899998, [151] := -2.919998, [152] := -2.939998, [153] := -2.959998, [154] := -2.9799979, [155] := -2.9999979, [156] := -3.0199978, [157] := -3.0399978, [158] := -3.0599978, [159] := -3.0799978, [160] := -3.0999978, [161] := -3.1199977, [162] := -3.1399977, [163] := -3.1599977, [164] := -3.1799977, [165] := -3.1999977, [166] := -3.2199976, [167] := -3.2399976, [168] := -3.2599976, [169] := -3.2799976, [170] := -3.2999976, [171] := -3.3199975, [172] := -3.3399975, [173] := -3.3599975, [174] := -3.3799975, [175] := -3.3999975, [176] := -3.4199975, [177] := -3.4399974, [178] := -3.4599974, [179] := -3.4799974, [180] := -3.4999974,
        [181] := -3.5199974, [182] := -3.5399973, [183] := -3.5599973, [184] := -3.5799973, [185] := -3.5999973, [186] := -3.6199973, [187] := -3.6399972, [188] := -3.6599972, [189] := -3.6799972, [190] := -3.6999972, [191] := -3.7199972, [192] := -3.7399971, [193] := -3.7599971, [194] := -3.779997, [195] := -3.799997, [196] := -3.819997, [197] := -3.839997, [198] := -3.859997, [199] := -3.879997, [200] := -3.899997, [201] := -3.919997, [202] := -3.939997, [203] := -3.959997, [204] := -3.979997, [205] := -3.999997, [206] := -4.019997, [207] := -4.039997, [208] := -4.059997, [209] := -4.079997, [210] := -4.099997, [211] := -4.119997, [212] := -4.139997, [213] := -4.159997, [214] := -4.179997, [215] := -4.199997, [216] := -4.219997, [217] := -4.239997, [218] := -4.259997, [219] := -4.279997, [220] := -4.299997, [221] := -4.319997, [222] := -4.339997, [223] := -4.359997, [224] := -4.379997, [225] := -4.3999968, [226] := -4.4199967, [227] := -4.4399967, [228] := -4.4599967, [229] := -4.4799967, [230] := -4.4999967, [231] := -4.5199966, [232] := -4.5399966, [233] := -4.5599966, [234] := -4.5799966, [235] := -4.5999966, [236] := -4.6199965, [237] := -4.6399965, [238] := -4.6599965, [239] := -4.6799965, [240] := -4.6999965,
        [241] := -4.7199965, [242] := -4.7399964, [243] := -4.7599964, [244] := -4.7799964, [245] := -4.7999964, [246] := -4.8199964, [247] := -4.8399963, [248] := -4.8599963, [249] := -4.8799963, [250] := -4.8999963, [251] := -4.9199963, [252] := -4.9399962, [253] := -4.959996, [254] := -4.979996, [255] := -4.999996, [256] := -5.019996, [257] := -5.039996, [258] := -5.059996, [259] := -5.079996, [260] := -5.099996, [261] := -5.119996, [262] := -5.139996, [263] := -5.159996, [264] := -5.179996, [265] := -5.199996, [266] := -5.219996, [267] := -5.239996, [268] := -5.259996, [269] := -5.279996, [270] := -5.299996, [271] := -5.319996, [272] := -5.339996, [273] := -5.359996, [274] := -5.379996, [275] := -5.399996, [276] := -5.419996, [277] := -5.439996, [278] := -5.4599957, [279] := -5.4799957, [280] := -5.4999957, [281] := -5.5199957, [282] := -5.5399957, [283] := -5.5599957, [284] := -5.5799956, [285] := -5.5999956, [286] := -5.6199956, [287] := -5.6399956, [288] := -5.6599956, [289] := -5.6799955, [290] := -5.6999955, [291] := -5.7199955, [292] := -5.7399955, [293] := -5.7599955, [294] := -5.7799954, [295] := -5.7999954, [296] := -5.8199954, [297] := -5.8399954, [298] := -5.8599954, [299] := -5.8799953, [300] := -5.8999953,
        [301] := -5.9199953, [302] := -5.9399953, [303] := -5.9599953, [304] := -5.9799953, [305] := -5.999995, [306] := -6.019995, [307] := -6.039995, [308] := -6.059995, [309] := -6.079995, [310] := -6.099995, [311] := -6.119995, [312] := -6.139995, [313] := -6.159995, [314] := -6.179995, [315] := -6.199995, [316] := -6.219995, [317] := -6.239995, [318] := -6.259995, [319] := -6.279995, [320] := -6.299995, [321] := -6.319995, [322] := -6.339995, [323] := -6.359995, [324] := -6.379995, [325] := -6.399995, [326] := -6.419995, [327] := -6.439995, [328] := -6.459995, [329] := -6.479995, [330] := -6.4999948, [331] := -6.5199947, [332] := -6.5399947, [333] := -6.5599947, [334] := -6.5799947, [335] := -6.5999947, [336] := -6.6199946, [337] := -6.6399946, [338] := -6.6599946, [339] := -6.6799946, [340] := -6.6999946, [341] := -6.7199945, [342] := -6.7399945, [343] := -6.7599945, [344] := -6.7799945, [345] := -6.7999945, [346] := -6.8199944, [347] := -6.8399944, [348] := -6.8599944, [349] := -6.8799944, [350] := -6.8999944, [351] := -6.9199944, [352] := -6.9399943, [353] := -6.9599943, [354] := -6.9799943, [355] := -6.9999943, [356] := -7.0199943, [357] := -7.0399942, [358] := -7.059994, [359] := -7.079994, [360] := -7.099994,
        [361] := -7.119994, [362] := -7.139994, [363] := -7.159994, [364] := -7.179994, [365] := -7.199994, [366] := -7.219994, [367] := -7.239994, [368] := -7.259994, [369] := -7.279994, [370] := -7.299994, [371] := -7.319994, [372] := -7.339994, [373] := -7.359994, [374] := -7.379994, [375] := -7.399994, [376] := -7.419994, [377] := -7.439994, [378] := -7.459994, [379] := -7.479994, [380] := -7.499994, [381] := -7.519994, [382] := -7.539994, [383] := -7.5599937, [384] := -7.5799937, [385] := -7.5999937, [386] := -7.6199937, [387] := -7.6399937, [388] := -7.6599936, [389] := -7.6799936, [390] := -7.6999936, [391] := -7.7199936, [392] := -7.7399936, [393] := -7.7599936, [394] := -7.7799935, [395] := -7.7999935, [396] := -7.8199935, [397] := -7.8399935, [398] := -7.8599935, [399] := -7.8799934, [400] := -7.8999934, [401] := -7.9199934, [402] := -7.9399934, [403] := -7.9599934, [404] := -7.9799933, [405] := -7.9999933, [406] := -8.019994, [407] := -8.039994, [408] := -8.059995, [409] := -8.079995, [410] := -8.099996, [411] := -8.119996, [412] := -8.139997, [413] := -8.159997, [414] := -8.179997, [415] := -8.199998, [416] := -8.219998, [417] := -8.239999, [418] := -8.259999, [419] := -8.28, [420] := -8.3,
        [421] := -8.320001, [422] := -8.340001, [423] := -8.360002, [424] := -8.380002, [425] := -8.4000025, [426] := -8.420003, [427] := -8.440003, [428] := -8.460004, [429] := -8.480004, [430] := -8.500005, [431] := -8.520005, [432] := -8.540006, [433] := -8.560006, [434] := -8.580007, [435] := -8.600007, [436] := -8.6200075, [437] := -8.640008, [438] := -8.660008, [439] := -8.680009, [440] := -8.700009, [441] := -8.72001, [442] := -8.74001, [443] := -8.760011, [444] := -8.780011, [445] := -8.800012, [446] := -8.820012, [447] := -8.840013, [448] := -8.860013, [449] := -8.880013, [450] := -8.900014, [451] := -8.920014, [452] := -8.940015, [453] := -8.960015, [454] := -8.980016, [455] := -9.000016, [456] := -9.020017, [457] := -9.040017, [458] := -9.060018, [459] := -9.080018, [460] := -9.1000185, [461] := -9.120019, [462] := -9.140019, [463] := -9.16002, [464] := -9.18002, [465] := -9.200021, [466] := -9.220021, [467] := -9.240022, [468] := -9.260022, [469] := -9.280023, [470] := -9.300023, [471] := -9.320024, [472] := -9.340024, [473] := -9.360024, [474] := -9.380025, [475] := -9.400025, [476] := -9.420026, [477] := -9.440026, [478] := -9.460027, [479] := -9.480027, [480] := -9.500028,
        [481] := -9.520028, [482] := -9.540029, [483] := -9.560029, [484] := -9.5800295, [485] := -9.60003, [486] := -9.62003, [487] := -9.640031, [488] := -9.660031, [489] := -9.680032, [490] := -9.700032, [491] := -9.720033, [492] := -9.740033, [493] := -9.760034, [494] := -9.780034, [495] := -9.8000345, [496] := -9.820035, [497] := -9.840035, [498] := -9.860036, [499] := -9.880036, [500] := -9.900037, [501] := -9.920037, [502] := -9.940038, [503] := -9.960038, [504] := -9.980039, [505] := -10.000039, [506] := -10.02004, [507] := -10.04004, [508] := -10.06004, [509] := -10.080041, [510] := -10.100041, [511] := -10.120042, [512] := -10.140042, [513] := -10.160043, [514] := -10.180043, [515] := -10.200044, [516] := -10.220044, [517] := -10.240045, [518] := -10.260045, [519] := -10.2800455, [520] := -10.300046, [521] := -10.320046, [522] := -10.340047, [523] := -10.360047, [524] := -10.380048, [525] := -10.400048, [526] := -10.420049, [527] := -10.440049, [528] := -10.46005, [529] := -10.48005, [530] := -10.500051, [531] := -10.520051, [532] := -10.540051, [533] := -10.560052, [534] := -10.580052, [535] := -10.600053, [536] := -10.620053, [537] := -10.640054, [538] := -10.660054, [539] := -10.680055, [540] := -10.700055,
        [541] := -10.720056, [542] := -10.740056, [543] := -10.7600565, [544] := -10.780057, [545] := -10.800057, [546] := -10.820058, [547] := -10.840058, [548] := -10.860059, [549] := -10.880059, [550] := -10.90006, [551] := -10.92006, [552] := -10.940061, [553] := -10.960061, [554] := -10.980062, [555] := -11.000062, [556] := -11.020062, [557] := -11.040063, [558] := -11.060063, [559] := -11.080064, [560] := -11.100064, [561] := -11.120065, [562] := -11.140065, [563] := -11.160066, [564] := -11.180066, [565] := -11.200067, [566] := -11.220067, [567] := -11.2400675, [568] := -11.260068, [569] := -11.280068, [570] := -11.300069, [571] := -11.320069, [572] := -11.34007, [573] := -11.36007, [574] := -11.380071, [575] := -11.400071, [576] := -11.420072, [577] := -11.440072, [578] := -11.4600725, [579] := -11.480073, [580] := -11.500073, [581] := -11.520074, [582] := -11.540074, [583] := -11.560075, [584] := -11.580075, [585] := -11.600076, [586] := -11.620076, [587] := -11.640077, [588] := -11.660077, [589] := -11.680078, [590] := -11.700078, [591] := -11.720078, [592] := -11.740079, [593] := -11.760079, [594] := -11.78008, [595] := -11.80008, [596] := -11.820081, [597] := -11.840081, [598] := -11.860082, [599] := -11.880082, [600] := -11.900083,
        [601] := -11.920083, [602] := -11.9400835, [603] := -11.960084, [604] := -11.980084, [605] := -12.000085, [606] := -12.020085, [607] := -12.040086, [608] := -12.060086, [609] := -12.080087, [610] := -12.100087, [611] := -12.120088, [612] := -12.140088, [613] := -12.160089, [614] := -12.180089, [615] := -12.200089, [616] := -12.22009, [617] := -12.24009, [618] := -12.260091, [619] := -12.280091, [620] := -12.300092, [621] := -12.320092, [622] := -12.340093, [623] := -12.360093, [624] := -12.380094, [625] := -12.400094, [626] := -12.4200945, [627] := -12.440095, [628] := -12.460095, [629] := -12.480096, [630] := -12.500096, [631] := -12.520097, [632] := -12.540097, [633] := -12.560098, [634] := -12.580098, [635] := -12.600099, [636] := -12.620099, [637] := -12.6401, [638] := -12.6601, [639] := -12.6801, [640] := -12.700101, [641] := -12.720101, [642] := -12.740102, [643] := -12.760102, [644] := -12.780103, [645] := -12.800103, [646] := -12.820104, [647] := -12.840104, [648] := -12.860105, [649] := -12.880105, [650] := -12.900105, [651] := -12.920106, [652] := -12.940106, [653] := -12.960107, [654] := -12.980107, [655] := -13.000108, [656] := -13.020108, [657] := -13.040109, [658] := -13.060109, [659] := -13.08011, [660] := -13.10011,
        [661] := -13.1201105, [662] := -13.140111, [663] := -13.160111, [664] := -13.180112, [665] := -13.200112, [666] := -13.220113, [667] := -13.240113, [668] := -13.260114, [669] := -13.280114, [670] := -13.300115, [671] := -13.320115, [672] := -13.340116, [673] := -13.360116, [674] := -13.380116, [675] := -13.400117, [676] := -13.420117, [677] := -13.440118, [678] := -13.460118, [679] := -13.480119, [680] := -13.500119, [681] := -13.52012, [682] := -13.54012, [683] := -13.560121, [684] := -13.580121, [685] := -13.6001215, [686] := -13.620122, [687] := -13.640122, [688] := -13.660123, [689] := -13.680123, [690] := -13.700124, [691] := -13.720124, [692] := -13.740125, [693] := -13.760125, [694] := -13.780126, [695] := -13.800126, [696] := -13.820127, [697] := -13.840127, [698] := -13.860127, [699] := -13.880128, [700] := -13.900128, [701] := -13.920129, [702] := -13.940129, [703] := -13.96013, [704] := -13.98013, [705] := -14.000131, [706] := -14.020131, [707] := -14.040132, [708] := -14.060132, [709] := -14.0801325, [710] := -14.100133, [711] := -14.120133, [712] := -14.140134, [713] := -14.160134, [714] := -14.180135, [715] := -14.200135, [716] := -14.220136, [717] := -14.240136, [718] := -14.260137, [719] := -14.280137, [720] := -14.3001375,
        [721] := -14.320138, [722] := -14.340138, [723] := -14.360139, [724] := -14.380139, [725] := -14.40014, [726] := -14.42014, [727] := -14.440141, [728] := -14.460141, [729] := -14.480142, [730] := -14.500142, [731] := -14.520143, [732] := -14.540143, [733] := -14.560143, [734] := -14.580144, [735] := -14.600144, [736] := -14.620145, [737] := -14.640145, [738] := -14.660146, [739] := -14.680146, [740] := -14.700147, [741] := -14.720147, [742] := -14.740148, [743] := -14.760148, [744] := -14.7801485, [745] := -14.800149, [746] := -14.820149, [747] := -14.84015, [748] := -14.86015, [749] := -14.880151, [750] := -14.900151, [751] := -14.920152, [752] := -14.940152, [753] := -14.960153, [754] := -14.980153, [755] := -15.000154, [756] := -15.020154, [757] := -15.040154, [758] := -15.060155, [759] := -15.080155, [760] := -15.100156, [761] := -15.120156, [762] := -15.140157, [763] := -15.160157, [764] := -15.180158, [765] := -15.200158, [766] := -15.220159, [767] := -15.240159, [768] := -15.2601595, [769] := -15.28016, [770] := -15.30016, [771] := -15.320161, [772] := -15.340161, [773] := -15.360162, [774] := -15.380162, [775] := -15.400163, [776] := -15.420163, [777] := -15.440164, [778] := -15.460164, [779] := -15.480165, [780] := -15.500165,
        [781] := -15.520165, [782] := -15.540166, [783] := -15.560166, [784] := -15.580167, [785] := -15.600167, [786] := -15.620168, [787] := -15.640168, [788] := -15.660169, [789] := -15.680169, [790] := -15.70017, [791] := -15.72017, [792] := -15.7401705, [793] := -15.760171, [794] := -15.780171, [795] := -15.800172, [796] := -15.820172, [797] := -15.840173, [798] := -15.860173, [799] := -0.1);
   QOP_HMI_GRAPH2_LINE1_DATAY : REAL[800] := ([0] := 4.251261, [1] := 4.251261, [2] := 4.251261, [3] := 4.251261, [4] := 4.251261, [5] := 4.251261, [6] := 4.251261, [7] := 4.251261, [8] := 4.251261, [9] := 4.251261, [10] := 4.251261, [11] := 4.251261, [12] := 4.251261, [13] := 4.251261, [14] := 4.251261, [15] := 4.251261, [16] := 4.251261, [17] := 4.251261, [18] := 4.251261, [19] := 4.251261, [20] := 4.251261, [21] := 4.251261, [22] := 4.251261, [23] := 4.251261, [24] := 4.251261, [25] := 4.251261, [26] := 4.251261, [27] := 4.251261, [28] := 4.251261, [29] := 4.251261, [30] := 4.251261, [31] := 4.251261, [32] := 4.251261, [33] := 4.251261, [34] := 4.251261, [35] := 4.251261, [36] := 4.251261, [37] := 4.251261, [38] := 4.251261, [39] := 4.251261, [40] := 4.251261, [41] := 4.251261, [42] := 4.251261, [43] := 4.251261, [44] := 4.251261, [45] := 4.251261, [46] := 4.251261, [47] := 4.251261, [48] := 4.251261, [49] := 4.251261, [50] := 4.251261, [51] := 4.251261, [52] := 4.251261, [53] := 4.251261, [54] := 4.251261, [55] := 5.1478252, [56] := 5.1478252, [57] := 5.1478252, [58] := 5.1478252, [59] := 5.1478252,
        [60] := 5.1478252, [61] := 5.1478252, [62] := 5.1478252, [63] := 5.1478252, [64] := 5.1478252, [65] := 5.1478252, [66] := 5.1478252, [67] := 5.1478252, [68] := 5.1478252, [69] := 5.1478252, [70] := 5.1478252, [71] := 5.1478252, [72] := 5.1478252, [73] := 5.1478252, [74] := 5.1478252, [75] := 5.1478252, [76] := 5.1478252, [77] := 5.1478252, [78] := 5.1478252, [79] := 5.1478252, [80] := 5.1478252, [81] := 5.1478252, [82] := 5.1478252, [83] := 5.1478252, [84] := 5.1478252, [85] := 5.1478252, [86] := 5.1478252, [87] := 5.1478252, [88] := 5.1478252, [89] := 5.1478252, [90] := 5.1478252, [91] := 5.1478252, [92] := 5.1478252, [93] := 5.1478252, [94] := 5.1478252, [95] := 5.1478252, [96] := 5.1478252, [97] := 5.1478252, [98] := 5.1478252, [99] := 5.1478252, [100] := 5.1478252, [101] := 5.1478252, [102] := 5.1478252, [103] := 5.1478252, [104] := 5.1478252, [105] := 5.1478252, [106] := 5.1478252, [107] := 5.1478252, [108] := 5.1478252, [109] := 5.1478252, [110] := 5.1478252, [111] := 5.1478252, [112] := 5.1478252, [113] := 5.3824944, [114] := 5.3824944, [115] := 5.3824944, [116] := 5.3824944, [117] := 5.3824944, [118] := 5.3824944, [119] := 5.3824944,
        [120] := 5.3824944, [121] := 5.3824944, [122] := 5.3824944, [123] := 5.3824944, [124] := 5.3824944, [125] := 5.3824944, [126] := 5.3824944, [127] := 5.3824944, [128] := 5.3824944, [129] := 5.3824944, [130] := 5.3824944, [131] := 5.3824944, [132] := 5.3824944, [133] := 5.3824944, [134] := 5.3824944, [135] := 5.3824944, [136] := 5.3824944, [137] := 5.3824944, [138] := 5.3824944, [139] := 5.3824944, [140] := 5.3824944, [141] := 5.3824944, [142] := 5.3824944, [143] := 5.3824944, [144] := 5.3824944, [145] := 5.3824944, [146] := 5.3824944, [147] := 5.3824944, [148] := 5.3824944, [149] := 5.3824944, [150] := 5.3824944, [151] := 5.3824944, [152] := 5.3824944, [153] := 5.3824944, [154] := 5.3824944, [155] := 4.5466924, [156] := 4.5466924, [157] := 4.5466924, [158] := 4.5466924, [159] := 4.5466924, [160] := 4.5466924, [161] := 4.5466924, [162] := 4.5466924, [163] := 4.5466924, [164] := 4.5466924, [165] := 4.5466924, [166] := 4.5466924, [167] := 4.5466924, [168] := 4.5466924, [169] := 4.5466924, [170] := 4.5466924, [171] := 4.5466924, [172] := 4.5466924, [173] := 4.5466924, [174] := 4.5466924, [175] := 4.5466924, [176] := 4.5466924, [177] := 4.5466924, [178] := 4.5466924, [179] := 4.5466924,
        [180] := 4.5466924, [181] := 4.5466924, [182] := 4.5466924, [183] := 4.5466924, [184] := 4.5466924, [185] := 4.5466924, [186] := 4.5466924, [187] := 4.5466924, [188] := 4.5466924, [189] := 4.5466924, [190] := 4.5466924, [191] := 4.5466924, [192] := 4.5466924, [193] := 4.5466924, [194] := 4.5466924, [195] := 4.5466924, [196] := 4.5466924, [197] := 4.5466924, [198] := 4.5466924, [199] := 4.5466924, [200] := 4.5466924, [201] := 4.5466924, [202] := 4.5466924, [203] := 4.5466924, [204] := 4.5466924, [205] := 4.5466924, [206] := 4.5466924, [207] := 4.5466924, [208] := 4.5466924, [209] := 4.5466924, [210] := 4.5466924, [211] := 3.9856725, [212] := 3.9856725, [213] := 3.9856725, [214] := 3.9856725, [215] := 3.9856725, [216] := 3.9856725, [217] := 3.9856725, [218] := 3.9856725, [219] := 3.9856725, [220] := 3.9856725, [221] := 3.9856725, [222] := 3.9856725, [223] := 3.9856725, [224] := 3.9856725, [225] := 3.9856725, [226] := 3.9856725, [227] := 3.9856725, [228] := 3.9856725, [229] := 3.9856725, [230] := 3.9856725, [231] := 3.9856725, [232] := 3.9856725, [233] := 3.9856725, [234] := 3.9856725, [235] := 3.9856725, [236] := 3.9856725, [237] := 3.9856725, [238] := 3.9856725, [239] := 3.9856725,
        [240] := 3.9856725, [241] := 3.9856725, [242] := 3.9856725, [243] := 3.9856725, [244] := 3.9856725, [245] := 3.9856725, [246] := 3.9856725, [247] := 3.9856725, [248] := 3.9856725, [249] := 3.9856725, [250] := 3.9856725, [251] := 3.9856725, [252] := 3.9856725, [253] := 3.9856725, [254] := 3.9856725, [255] := 3.9856725, [256] := 3.9856725, [257] := 3.9856725, [258] := 3.9856725, [259] := 3.9856725, [260] := 3.9856725, [261] := 3.9856725, [262] := 3.9856725, [263] := 3.9856725, [264] := 3.9856725, [265] := 3.9856725, [266] := 3.9856725, [267] := 3.9856725, [268] := 4.2594185, [269] := 4.2594185, [270] := 4.2594185, [271] := 4.2594185, [272] := 4.2594185, [273] := 4.2594185, [274] := 4.2594185, [275] := 4.2594185, [276] := 4.2594185, [277] := 4.2594185, [278] := 4.2594185, [279] := 4.2594185, [280] := 4.2594185, [281] := 4.2594185, [282] := 4.2594185, [283] := 4.2594185, [284] := 4.2594185, [285] := 4.2594185, [286] := 4.2594185, [287] := 4.2594185, [288] := 4.2594185, [289] := 4.2594185, [290] := 4.2594185, [291] := 4.2594185, [292] := 4.2594185, [293] := 4.2594185, [294] := 4.2594185, [295] := 4.2594185, [296] := 4.2594185, [297] := 4.2594185, [298] := 4.2594185, [299] := 4.2594185,
        [300] := 4.2594185, [301] := 4.2594185, [302] := 4.2594185, [303] := 4.2594185, [304] := 4.2594185, [305] := 4.2594185, [306] := 4.2594185, [307] := 4.2594185, [308] := 4.2594185, [309] := 4.2594185, [310] := 4.2594185, [311] := 4.2594185, [312] := 4.2594185, [313] := 4.2594185, [314] := 4.2594185, [315] := 4.2594185, [316] := 4.2594185, [317] := 4.2594185, [318] := 4.2594185, [319] := 4.2594185, [320] := 4.2594185, [321] := 4.2594185, [322] := 4.2594185, [323] := 4.2594185, [324] := 4.2594185, [325] := 4.2594185, [326] := 3.9511158, [327] := 3.9511158, [328] := 3.9511158, [329] := 3.9511158, [330] := 3.9511158, [331] := 3.9511158, [332] := 3.9511158, [333] := 3.9511158, [334] := 3.9511158, [335] := 3.9511158, [336] := 3.9511158, [337] := 3.9511158, [338] := 3.9511158, [339] := 3.9511158, [340] := 3.9511158, [341] := 3.9511158, [342] := 3.9511158, [343] := 3.9511158, [344] := 3.9511158, [345] := 3.9511158, [346] := 3.9511158, [347] := 3.9511158, [348] := 3.9511158, [349] := 3.9511158, [350] := 3.9511158, [351] := 3.9511158, [352] := 3.9511158, [353] := 3.9511158, [354] := 3.9511158, [355] := 3.9511158, [356] := 3.9511158, [357] := 3.9511158, [358] := 3.9511158, [359] := 3.9511158,
        [360] := 3.9511158, [361] := 3.9511158, [362] := 3.9511158, [363] := 3.9511158, [364] := 3.9511158, [365] := 3.9511158, [366] := 3.9511158, [367] := 3.9511158, [368] := 3.9511158, [369] := 3.9511158, [370] := 3.9511158, [371] := 3.9511158, [372] := 3.9511158, [373] := 3.9511158, [374] := 3.9511158, [375] := 3.9511158, [376] := 3.9511158, [377] := 3.9511158, [378] := 3.9511158, [379] := 3.9511158, [380] := 3.9511158, [381] := 3.9511158, [382] := 5.4046583, [383] := 5.4046583, [384] := 5.4046583, [385] := 5.4046583, [386] := 5.4046583, [387] := 5.4046583, [388] := 5.4046583, [389] := 5.4046583, [390] := 5.4046583, [391] := 5.4046583, [392] := 5.4046583, [393] := 5.4046583, [394] := 5.4046583, [395] := 5.4046583, [396] := 5.4046583, [397] := 5.4046583, [398] := 5.4046583, [399] := 5.4046583, [400] := 5.4046583, [401] := 5.4046583, [402] := 5.4046583, [403] := 5.4046583, [404] := 5.4046583, [405] := 5.4046583, [406] := 5.4046583, [407] := 5.4046583, [408] := 5.4046583, [409] := 5.4046583, [410] := 5.4046583, [411] := 5.4046583, [412] := 5.4046583, [413] := 5.4046583, [414] := 5.4046583, [415] := 5.4046583, [416] := 5.4046583, [417] := 5.4046583, [418] := 5.4046583, [419] := 5.4046583,
        [420] := 5.4046583, [421] := 5.4046583, [422] := 5.4046583, [423] := 5.4046583, [424] := 5.4046583, [425] := 5.4046583, [426] := 5.4046583, [427] := 5.4046583, [428] := 5.4046583, [429] := 5.4046583, [430] := 5.4046583, [431] := 5.4046583, [432] := 5.4046583, [433] := 5.4046583, [434] := 5.4046583, [435] := 5.4046583, [436] := 5.4046583, [437] := 5.4046583, [438] := 5.4046583, [439] := 4.020748, [440] := 4.020748, [441] := 4.020748, [442] := 4.020748, [443] := 4.020748, [444] := 4.020748, [445] := 4.020748, [446] := 4.020748, [447] := 4.020748, [448] := 4.020748, [449] := 4.020748, [450] := 4.020748, [451] := 4.020748, [452] := 4.020748, [453] := 4.020748, [454] := 4.020748, [455] := 4.020748, [456] := 4.020748, [457] := 4.020748, [458] := 4.020748, [459] := 4.020748, [460] := 4.020748, [461] := 4.020748, [462] := 4.020748, [463] := 4.020748, [464] := 4.020748, [465] := 4.020748, [466] := 4.020748, [467] := 4.020748, [468] := 4.020748, [469] := 4.020748, [470] := 4.020748, [471] := 4.020748, [472] := 4.020748, [473] := 4.020748, [474] := 4.020748, [475] := 4.020748, [476] := 4.020748, [477] := 4.020748, [478] := 4.020748, [479] := 4.020748,
        [480] := 4.020748, [481] := 4.020748, [482] := 4.020748, [483] := 4.020748, [484] := 4.020748, [485] := 4.020748, [486] := 4.020748, [487] := 4.020748, [488] := 4.020748, [489] := 4.020748, [490] := 4.020748, [491] := 4.020748, [492] := 4.020748, [493] := 4.020748, [494] := 4.020748, [495] := 4.020748, [496] := 4.2406282, [497] := 4.2406282, [498] := 4.2406282, [499] := 4.2406282, [500] := 4.2406282, [501] := 4.2406282, [502] := 4.2406282, [503] := 4.2406282, [504] := 4.2406282, [505] := 4.2406282, [506] := 4.2406282, [507] := 4.2406282, [508] := 4.2406282, [509] := 4.2406282, [510] := 4.2406282, [511] := 4.2406282, [512] := 4.2406282, [513] := 4.2406282, [514] := 4.2406282, [515] := 4.2406282, [516] := 4.2406282, [517] := 4.2406282, [518] := 4.2406282, [519] := 4.2406282, [520] := 4.2406282, [521] := 4.2406282, [522] := 4.2406282, [523] := 4.2406282, [524] := 4.2406282, [525] := 4.2406282, [526] := 4.2406282, [527] := 4.2406282, [528] := 4.2406282, [529] := 4.2406282, [530] := 4.2406282, [531] := 4.2406282, [532] := 4.2406282, [533] := 4.2406282, [534] := 4.2406282, [535] := 4.2406282, [536] := 4.2406282, [537] := 4.2406282, [538] := 4.2406282, [539] := 4.2406282,
        [540] := 4.2406282, [541] := 4.2406282, [542] := 4.2406282, [543] := 4.2406282, [544] := 4.2406282, [545] := 4.2406282, [546] := 4.2406282, [547] := 4.2406282, [548] := 4.2406282, [549] := 4.2406282, [550] := 4.2406282, [551] := 4.2406282, [552] := 4.2406282, [553] := 4.53066, [554] := 4.53066, [555] := 4.53066, [556] := 4.53066, [557] := 4.53066, [558] := 4.53066, [559] := 4.53066, [560] := 4.53066, [561] := 4.53066, [562] := 4.53066, [563] := 4.53066, [564] := 4.53066, [565] := 4.53066, [566] := 4.53066, [567] := 4.53066, [568] := 4.53066, [569] := 4.53066, [570] := 4.53066, [571] := 4.53066, [572] := 4.53066, [573] := 4.53066, [574] := 4.53066, [575] := 4.53066, [576] := 4.53066, [577] := 4.53066, [578] := 4.53066, [579] := 4.53066, [580] := 4.53066, [581] := 4.53066, [582] := 4.53066, [583] := 4.53066, [584] := 4.53066, [585] := 4.53066, [586] := 4.53066, [587] := 4.53066, [588] := 4.53066, [589] := 4.53066, [590] := 4.53066, [591] := 4.53066, [592] := 4.53066, [593] := 4.53066, [594] := 4.53066, [595] := 4.53066, [596] := 4.53066, [597] := 4.53066, [598] := 4.53066, [599] := 4.53066,
        [600] := 4.53066, [601] := 4.53066, [602] := 4.53066, [603] := 4.53066, [604] := 4.53066, [605] := 4.53066, [606] := 4.53066, [607] := 4.53066, [608] := 4.53066, [609] := 4.53066, [610] := 4.53066, [611] := 5.2263255, [612] := 5.2263255, [613] := 5.2263255, [614] := 5.2263255, [615] := 5.2263255, [616] := 5.2263255, [617] := 5.2263255, [618] := 5.2263255, [619] := 5.2263255, [620] := 5.2263255, [621] := 5.2263255, [622] := 5.2263255, [623] := 5.2263255, [624] := 5.2263255, [625] := 5.2263255, [626] := 5.2263255, [627] := 5.2263255, [628] := 5.2263255, [629] := 5.2263255, [630] := 5.2263255, [631] := 5.2263255, [632] := 5.2263255, [633] := 5.2263255, [634] := 5.2263255, [635] := 5.2263255, [636] := 5.2263255, [637] := 5.2263255, [638] := 5.2263255, [639] := 5.2263255, [640] := 5.2263255, [641] := 5.2263255, [642] := 5.2263255, [643] := 5.2263255, [644] := 5.2263255, [645] := 5.2263255, [646] := 5.2263255, [647] := 5.2263255, [648] := 5.2263255, [649] := 5.2263255, [650] := 5.2263255, [651] := 5.2263255, [652] := 5.2263255, [653] := 5.2263255, [654] := 5.2263255, [655] := 5.2263255, [656] := 5.2263255, [657] := 5.2263255, [658] := 5.2263255, [659] := 5.2263255,
        [660] := 5.2263255, [661] := 5.2263255, [662] := 5.2263255, [663] := 5.2263255, [664] := 5.2263255, [665] := 5.2263255, [666] := 5.2263255, [667] := 5.2263255, [668] := 3.9186366, [669] := 3.9186366, [670] := 3.9186366, [671] := 3.9186366, [672] := 3.9186366, [673] := 3.9186366, [674] := 3.9186366, [675] := 3.9186366, [676] := 3.9186366, [677] := 3.9186366, [678] := 3.9186366, [679] := 3.9186366, [680] := 3.9186366, [681] := 3.9186366, [682] := 3.9186366, [683] := 3.9186366, [684] := 3.9186366, [685] := 3.9186366, [686] := 3.9186366, [687] := 3.9186366, [688] := 3.9186366, [689] := 3.9186366, [690] := 3.9186366, [691] := 3.9186366, [692] := 3.9186366, [693] := 3.9186366, [694] := 3.9186366, [695] := 3.9186366, [696] := 3.9186366, [697] := 3.9186366, [698] := 3.9186366, [699] := 3.9186366, [700] := 3.9186366, [701] := 3.9186366, [702] := 3.9186366, [703] := 3.9186366, [704] := 3.9186366, [705] := 3.9186366, [706] := 3.9186366, [707] := 3.9186366, [708] := 3.9186366, [709] := 3.9186366, [710] := 3.9186366, [711] := 4.232493, [712] := 4.232493, [713] := 4.232493, [714] := 4.232493, [715] := 4.232493, [716] := 4.232493, [717] := 4.232493, [718] := 4.232493, [719] := 4.232493,
        [720] := 4.232493, [721] := 4.232493, [722] := 4.232493, [723] := 4.232493, [724] := 4.232493, [725] := 4.232493, [726] := 4.232493, [727] := 4.232493, [728] := 4.232493, [729] := 4.232493, [730] := 4.232493, [731] := 4.232493, [732] := 4.232493, [733] := 4.232493, [734] := 4.232493, [735] := 4.232493, [736] := 4.232493, [737] := 4.232493, [738] := 4.232493, [739] := 4.232493, [740] := 4.232493, [741] := 4.232493, [742] := 4.232493, [743] := 4.232493, [744] := 4.232493, [745] := 4.232493, [746] := 4.232493, [747] := 4.232493, [748] := 4.232493, [749] := 4.232493, [750] := 4.232493, [751] := 4.232493, [752] := 4.232493, [753] := 4.232493, [754] := 4.232493, [755] := 4.232493, [756] := 4.232493, [757] := 4.232493, [758] := 4.232493, [759] := 4.232493, [760] := 4.232493, [761] := 4.232493, [762] := 4.232493, [763] := 4.232493, [764] := 4.232493, [765] := 4.232493, [766] := 4.232493, [767] := 3.4168825, [768] := 3.4168825, [769] := 3.4168825, [770] := 3.4168825, [771] := 3.4168825, [772] := 3.4168825, [773] := 3.4168825, [774] := 3.4168825, [775] := 3.4168825, [776] := 3.4168825, [777] := 3.4168825, [778] := 3.4168825, [779] := 3.4168825,
        [780] := 3.4168825, [781] := 3.4168825, [782] := 3.4168825, [783] := 3.4168825, [784] := 3.4168825, [785] := 3.4168825, [786] := 3.4168825, [787] := 3.4168825, [788] := 3.4168825, [789] := 3.4168825, [790] := 3.4168825, [791] := 3.4168825, [792] := 3.4168825, [793] := 3.4168825, [794] := 3.4168825, [795] := 3.4168825, [796] := 3.4168825, [797] := 3.4168825, [798] := 3.4168825, [799] := 3.4168825);
   QOP_HMI_GRAPH2_LINE1_HDR : REAL[10] := ([0] := 800.0, [4] := 1.0);
   QOP_HMI_GRAPH2_LINE2_DATAY : REAL[800];
   QOP_HMI_REAL : REAL[20] := ([3] := 10000.0, [4] := -357.83133, [5] := 357.83133);
   RondjesT1 : REAL := 40.0;
   RondjesT2 : REAL;
   SAF_RESET_KNOP : BOOL;
   Safeovertravel1 : REAL := -0.001; {access None}
   Safeovertravel2 : REAL := 0.004; {access None}
   SAFETY_DOOR1_OPEN : BOOL;
   SAFETY_DOOR2_OPEN : BOOL;
   Start_testrun1 : BOOL;
   StartG : ALIAS FOR RIO_CTRL:3:I.0;
   StartLampje : ALIAS FOR RIO_CTRL:5:O.0;
   StartT1 : ALIAS FOR IOP_HMI_BT[0].0;
   StartT2 : ALIAS FOR IOP_HMI_BT[1].0;
   StateT1Routine : DINT;
   StateT2Routine : DINT := 62;
